LIN {X 0.002,Y -301.085,Z 1918.358,A 0.000,B 0.000,C 90.000,E1 64.357} C_DIS
LIN {X -0.093,Y -288.986,Z 1918.341,A 0.000,B 0.000,C 90.000,E1 61.385} C_DIS
LIN {X 0.024,Y -280.949,Z 1918.330,A 0.000,B 0.000,C 90.000,E1 59.331} C_DIS
LIN {X 0.071,Y -271.438,Z 1918.316,A 0.000,B 0.000,C 90.000,E1 56.914} C_DIS
LIN {X 0.067,Y -263.244,Z 1918.305,A 0.000,B 0.000,C 90.000,E1 54.815} C_DIS
LIN {X -0.054,Y -253.623,Z 1918.291,A 0.000,B 0.000,C 90.000,E1 52.351} C_DIS
LIN {X -0.111,Y -244.044,Z 1918.277,A 0.000,B 0.000,C 90.000,E1 49.828} C_DIS
LIN {X 0.069,Y -233.329,Z 1918.260,A 0.000,B 0.000,C 90.000,E1 46.824} C_DIS
LIN {X 0.121,Y -223.019,Z 1918.243,A 0.000,B 0.000,C 90.000,E1 43.785} C_DIS
LIN {X 0.001,Y -212.058,Z 1918.224,A 0.000,B 0.000,C 90.000,E1 40.334} C_DIS
LIN {X 0.010,Y -204.184,Z 1918.209,A 0.000,B 0.000,C 90.000,E1 37.569} C_DIS
LIN {X 0.020,Y -196.023,Z 1918.191,A 0.000,B 0.000,C 90.000,E1 34.358} C_DIS
LIN {X -0.106,Y -188.602,Z 1918.173,A 0.000,B 0.000,C 90.000,E1 31.131} C_DIS
LIN {X 0.030,Y -181.908,Z 1918.154,A 0.000,B 0.000,C 90.000,E1 27.769} C_DIS
LIN {X 0.067,Y -175.929,Z 1918.136,A 0.000,B 0.000,C 90.000,E1 24.387} C_DIS
LIN {X 0.063,Y -170.772,Z 1918.117,A 0.000,B 0.000,C 90.000,E1 20.972} C_DIS
LIN {X 0.072,Y -166.432,Z 1918.097,A 0.000,B 0.000,C 90.000,E1 17.511} C_DIS
LIN {X -0.056,Y -162.887,Z 1918.078,A 0.000,B 0.000,C 90.000,E1 14.064} C_DIS
LIN {X -0.062,Y -159.922,Z 1918.058,A 0.000,B 0.000,C 90.000,E1 10.546} C_DIS
LIN {X 0.005,Y -157.280,Z 1918.034,A 0.000,B 0.000,C 90.000,E1 6.087} C_DIS
LIN {X 0.000,Y -154.958,Z 1918.000,A 0.000,B 0.000,C 90.000,E1 360.000} C_DIS
LIN {X 0.053,Y -154.095,Z 1917.953,A 0.000,B 0.000,C 90.000,E1 351.432} C_DIS
LIN {X -0.028,Y -155.826,Z 1917.913,A 0.000,B 0.000,C 90.000,E1 344.283} C_DIS
LIN {X 0.033,Y -158.560,Z 1917.883,A 0.000,B 0.000,C 90.000,E1 338.901} C_DIS
LIN {X 0.047,Y -162.161,Z 1917.858,A 0.000,B 0.000,C 90.000,E1 334.460} C_DIS
LIN {X -0.046,Y -166.070,Z 1917.839,A 0.000,B 0.000,C 90.000,E1 330.973} C_DIS
LIN {X 0.051,Y -170.958,Z 1917.819,A 0.000,B 0.000,C 90.000,E1 327.454} C_DIS
LIN {X -0.037,Y -175.264,Z 1917.805,A 0.000,B 0.000,C 90.000,E1 324.895} C_DIS
LIN {X 0.017,Y -180.240,Z 1917.791,A 0.000,B 0.000,C 90.000,E1 322.316} C_DIS
LIN {X 0.016,Y -186.100,Z 1917.777,A 0.000,B 0.000,C 90.000,E1 319.784} C_DIS
LIN {X -0.018,Y -191.710,Z 1917.765,A 0.000,B 0.000,C 90.000,E1 317.715} C_DIS
LIN {X 0.020,Y -199.361,Z 1917.751,A 0.000,B 0.000,C 90.000,E1 315.243} C_DIS
LIN {X -0.078,Y -207.953,Z 1917.738,A 0.000,B 0.000,C 90.000,E1 312.852} C_DIS
LIN {X -0.098,Y -219.024,Z 1917.723,A 0.000,B 0.000,C 90.000,E1 310.092} C_DIS
LIN {X 0.025,Y -231.136,Z 1917.708,A 0.000,B 0.000,C 90.000,E1 307.363} C_DIS
LIN {X -0.158,Y -246.074,Z 1917.691,A 0.000,B 0.000,C 90.000,E1 304.405} C_DIS
LIN {X -0.153,Y -257.927,Z 1917.679,A 0.000,B 0.000,C 90.000,E1 302.212} C_DIS
LIN {X 0.088,Y -272.002,Z 1917.665,A 0.000,B 0.000,C 90.000,E1 299.667} C_DIS
LIN {X -0.137,Y -281.893,Z 1917.655,A 0.000,B 0.000,C 90.000,E1 297.975} C_DIS
LIN {X 0.036,Y -291.493,Z 1917.646,A 0.000,B 0.000,C 90.000,E1 296.232} C_DIS
LIN {X 0.116,Y -296.930,Z 1917.640,A 0.000,B 0.000,C 90.000,E1 295.207} C_DIS
LIN {X 0.120,Y -301.742,Z 1917.635,A 0.000,B 0.000,C 90.000,E1 294.207} C_DIS
LIN {X 0.005,Y -304.537,Z 1917.631,A 0.000,B 0.000,C 90.000,E1 293.567} C_DIS
LIN {X 0.067,Y -306.941,Z 1917.627,A 0.000,B 0.000,C 90.000,E1 292.898} C_DIS
LIN {X -0.019,Y -308.963,Z 1917.624,A 0.000,B 0.000,C 90.000,E1 292.259} C_DIS
LIN {X 0.070,Y -310.637,Z 1917.620,A 0.000,B 0.000,C 90.000,E1 291.589} C_DIS
LIN {X -0.116,Y -311.978,Z 1917.616,A 0.000,B 0.000,C 90.000,E1 290.972} C_DIS
LIN {X -0.001,Y -312.989,Z 1917.613,A 0.000,B 0.000,C 90.000,E1 290.301} C_DIS
LIN {X 0.124,Y -313.630,Z 1917.609,A 0.000,B 0.000,C 90.000,E1 289.631} C_DIS
LIN {X 0.145,Y -313.979,Z 1917.605,A 0.000,B 0.000,C 90.000,E1 288.960} C_DIS
LIN {X 0.090,Y -315.398,Z 1917.605,A 0.000,B 0.000,C 90.000,E1 288.960} C_DIS
LIN {X 0.111,Y -317.051,Z 1917.605,A 0.000,B 0.000,C 90.000,E1 288.906} C_DIS
LIN {X 0.074,Y -321.018,Z 1917.604,A 0.000,B 0.000,C 90.000,E1 288.671} C_DIS
LIN {X -0.008,Y -324.781,Z 1917.602,A 0.000,B 0.000,C 90.000,E1 288.362} C_DIS
LIN {X -0.038,Y -329.523,Z 1917.599,A 0.000,B 0.000,C 90.000,E1 287.873} C_DIS
LIN {X 0.007,Y -334.337,Z 1917.596,A 0.000,B 0.000,C 90.000,E1 287.275} C_DIS
LIN {X -0.155,Y -338.741,Z 1917.593,A 0.000,B 0.000,C 90.000,E1 286.677} C_DIS
LIN {X 0.038,Y -342.538,Z 1917.589,A 0.000,B 0.000,C 90.000,E1 286.024} C_DIS
LIN {X -0.073,Y -345.806,Z 1917.586,A 0.000,B 0.000,C 90.000,E1 285.426} C_DIS
LIN {X 0.173,Y -348.683,Z 1917.582,A 0.000,B 0.000,C 90.000,E1 284.773} C_DIS
LIN {X 0.027,Y -352.297,Z 1917.577,A 0.000,B 0.000,C 90.000,E1 283.883} C_DIS
LIN {X -0.172,Y -354.899,Z 1917.572,A 0.000,B 0.000,C 90.000,E1 283.008} C_DIS
LIN {X 0.132,Y -356.054,Z 1917.569,A 0.000,B 0.000,C 90.000,E1 282.355} C_DIS
LIN {X 0.021,Y -356.751,Z 1917.565,A 0.000,B 0.000,C 90.000,E1 281.771} C_DIS
LIN {X -0.083,Y -356.912,Z 1917.562,A 0.000,B 0.000,C 90.000,E1 281.186} C_DIS
LIN {X 0.169,Y -356.637,Z 1917.559,A 0.000,B 0.000,C 90.000,E1 280.546} C_DIS
LIN {X 0.070,Y -355.925,Z 1917.555,A 0.000,B 0.000,C 90.000,E1 279.962} C_DIS
LIN {X -0.032,Y -354.775,Z 1917.552,A 0.000,B 0.000,C 90.000,E1 279.378} C_DIS
LIN {X 0.155,Y -353.206,Z 1917.549,A 0.000,B 0.000,C 90.000,E1 278.746} C_DIS
LIN {X 0.041,Y -351.190,Z 1917.545,A 0.000,B 0.000,C 90.000,E1 278.163} C_DIS
LIN {X -0.132,Y -348.661,Z 1917.542,A 0.000,B 0.000,C 90.000,E1 277.587} C_DIS
LIN {X 0.066,Y -345.529,Z 1917.539,A 0.000,B 0.000,C 90.000,E1 276.947} C_DIS
LIN {X -0.056,Y -343.742,Z 1917.537,A 0.000,B 0.000,C 90.000,E1 276.663} C_DIS
LIN {X 0.071,Y -339.329,Z 1917.534,A 0.000,B 0.000,C 90.000,E1 276.030} C_DIS
LIN {X -0.022,Y -336.617,Z 1917.532,A 0.000,B 0.000,C 90.000,E1 275.739} C_DIS
LIN {X -0.082,Y -333.609,Z 1917.530,A 0.000,B 0.000,C 90.000,E1 275.448} C_DIS
LIN {X 0.158,Y -330.113,Z 1917.529,A 0.000,B 0.000,C 90.000,E1 275.106} C_DIS
LIN {X 0.053,Y -326.707,Z 1917.527,A 0.000,B 0.000,C 90.000,E1 274.878} C_DIS
LIN {X 0.082,Y -320.483,Z 1917.525,A 0.000,B 0.000,C 90.000,E1 274.531} C_DIS
LIN {X 0.041,Y -317.170,Z 1917.525,A 0.000,B 0.000,C 90.000,E1 274.416} C_DIS
LIN {X -0.141,Y -312.787,Z 1917.524,A 0.000,B 0.000,C 90.000,E1 274.359} C_DIS
LIN {X 0.063,Y -181.047,Z 1917.524,A 0.000,B 0.000,C 90.000,E1 274.302} C_DIS
LIN {X 0.057,Y -181.570,Z 1917.500,A 0.000,B 0.000,C 90.000,E1 270.057} C_DIS
LIN {X 0.044,Y -180.866,Z 1917.472,A 0.000,B 0.000,C 90.000,E1 265.008} C_DIS
LIN {X -0.078,Y -178.981,Z 1917.444,A 0.000,B 0.000,C 90.000,E1 259.982} C_DIS
LIN {X -0.067,Y -177.953,Z 1917.435,A 0.000,B 0.000,C 90.000,E1 258.285} C_DIS
LIN {X -0.048,Y -175.594,Z 1917.411,A 0.000,B 0.000,C 90.000,E1 254.031} C_DIS
LIN {X -0.035,Y -172.318,Z 1917.387,A 0.000,B 0.000,C 90.000,E1 249.752} C_DIS
LIN {X -0.056,Y -171.797,Z 1917.383,A 0.000,B 0.000,C 90.000,E1 248.901} C_DIS
LIN {X -0.019,Y -169.468,Z 1917.368,A 0.000,B 0.000,C 90.000,E1 246.305} C_DIS
LIN {X 0.037,Y -166.796,Z 1917.349,A 0.000,B 0.000,C 90.000,E1 242.820} C_DIS
LIN {X 0.032,Y -162.777,Z 1917.325,A 0.000,B 0.000,C 90.000,E1 238.456} C_DIS
LIN {X 0.008,Y -161.466,Z 1917.315,A 0.000,B 0.000,C 90.000,E1 236.707} C_DIS
LIN {X 0.049,Y -157.460,Z 1917.291,A 0.000,B 0.000,C 90.000,E1 232.271} C_DIS
LIN {X -0.018,Y -155.472,Z 1917.276,A 0.000,B 0.000,C 90.000,E1 229.622} C_DIS
LIN {X -0.085,Y -151.784,Z 1917.251,A 0.000,B 0.000,C 90.000,E1 225.162} C_DIS
LIN {X -0.071,Y -149.990,Z 1917.236,A 0.000,B 0.000,C 90.000,E1 222.447} C_DIS
LIN {X -0.040,Y -146.822,Z 1917.210,A 0.000,B 0.000,C 90.000,E1 217.890} C_DIS
LIN {X 0.066,Y -145.401,Z 1917.195,A 0.000,B 0.000,C 90.000,E1 215.105} C_DIS
LIN {X -0.017,Y -142.835,Z 1917.170,A 0.000,B 0.000,C 90.000,E1 210.541} C_DIS
LIN {X 0.040,Y -141.447,Z 1917.149,A 0.000,B 0.000,C 90.000,E1 206.821} C_DIS
LIN {X -0.047,Y -139.371,Z 1917.113,A 0.000,B 0.000,C 90.000,E1 200.355} C_DIS
LIN {X 0.070,Y -138.819,Z 1917.097,A 0.000,B 0.000,C 90.000,E1 197.511} C_DIS
LIN {X -0.016,Y -138.352,Z 1917.056,A 0.000,B 0.000,C 90.000,E1 190.074} C_DIS
LIN {X -0.043,Y -139.535,Z 1917.004,A 0.000,B 0.000,C 90.000,E1 180.745} C_DIS
LIN {X 0.051,Y -141.221,Z 1916.973,A 0.000,B 0.000,C 90.000,E1 175.122} C_DIS
LIN {X 0.009,Y -142.594,Z 1916.958,A 0.000,B 0.000,C 90.000,E1 172.356} C_DIS
LIN {X -0.038,Y -144.896,Z 1916.932,A 0.000,B 0.000,C 90.000,E1 167.757} C_DIS
LIN {X -0.084,Y -147.525,Z 1916.911,A 0.000,B 0.000,C 90.000,E1 164.102} C_DIS
LIN {X -0.010,Y -150.120,Z 1916.891,A 0.000,B 0.000,C 90.000,E1 160.423} C_DIS
LIN {X 0.001,Y -153.482,Z 1916.871,A 0.000,B 0.000,C 90.000,E1 156.794} C_DIS
LIN {X 0.065,Y -157.847,Z 1916.846,A 0.000,B 0.000,C 90.000,E1 152.281} C_DIS
LIN {X 0.021,Y -162.132,Z 1916.826,A 0.000,B 0.000,C 90.000,E1 148.742} C_DIS
LIN {X 0.000,Y -166.335,Z 1916.807,A 0.000,B 0.000,C 90.000,E1 145.229} C_DIS
LIN {X 0.007,Y -171.352,Z 1916.787,A 0.000,B 0.000,C 90.000,E1 141.743} C_DIS
LIN {X -0.066,Y -176.258,Z 1916.768,A 0.000,B 0.000,C 90.000,E1 138.324} C_DIS
LIN {X 0.052,Y -180.540,Z 1916.754,A 0.000,B 0.000,C 90.000,E1 135.729} C_DIS
LIN {X 0.032,Y -185.942,Z 1916.735,A 0.000,B 0.000,C 90.000,E1 132.366} C_DIS
LIN {X -0.033,Y -190.572,Z 1916.722,A 0.000,B 0.000,C 90.000,E1 129.886} C_DIS
LIN {X -0.003,Y -196.322,Z 1916.703,A 0.000,B 0.000,C 90.000,E1 126.583} C_DIS
LIN {X 0.075,Y -201.120,Z 1916.690,A 0.000,B 0.000,C 90.000,E1 124.119} C_DIS
LIN {X -0.006,Y -207.058,Z 1916.672,A 0.000,B 0.000,C 90.000,E1 120.924} C_DIS
LIN {X -0.010,Y -210.341,Z 1916.663,A 0.000,B 0.000,C 90.000,E1 119.333} C_DIS
LIN {X -0.016,Y -216.123,Z 1916.645,A 0.000,B 0.000,C 90.000,E1 116.181} C_DIS
LIN {X -0.112,Y -219.295,Z 1916.637,A 0.000,B 0.000,C 90.000,E1 114.643} C_DIS
LIN {X -0.109,Y -224.163,Z 1916.621,A 0.000,B 0.000,C 90.000,E1 111.844} C_DIS
LIN {X -0.174,Y -283.727,Z 1916.621,A 0.000,B 0.000,C 90.000,E1 111.844} C_DIS
LIN {X -0.106,Y -286.571,Z 1916.621,A 0.000,B 0.000,C 90.000,E1 111.770} C_DIS
LIN {X -0.081,Y -290.600,Z 1916.620,A 0.000,B 0.000,C 90.000,E1 111.535} C_DIS
LIN {X 0.088,Y -294.035,Z 1916.618,A 0.000,B 0.000,C 90.000,E1 111.153} C_DIS
LIN {X -0.092,Y -297.648,Z 1916.614,A 0.000,B 0.000,C 90.000,E1 110.610} C_DIS
LIN {X -0.075,Y -311.022,Z 1916.602,A 0.000,B 0.000,C 90.000,E1 108.290} C_DIS
LIN {X -0.041,Y -325.770,Z 1916.589,A 0.000,B 0.000,C 90.000,E1 106.024} C_DIS
LIN {X 0.046,Y -339.604,Z 1916.578,A 0.000,B 0.000,C 90.000,E1 104.120} C_DIS
LIN {X -0.103,Y -354.634,Z 1916.568,A 0.000,B 0.000,C 90.000,E1 102.299} C_DIS
LIN {X 0.070,Y -373.070,Z 1916.557,A 0.000,B 0.000,C 90.000,E1 100.254} C_DIS
LIN {X -0.187,Y -391.979,Z 1916.547,A 0.000,B 0.000,C 90.000,E1 98.454} C_DIS
LIN {X -0.144,Y -411.225,Z 1916.538,A 0.000,B 0.000,C 90.000,E1 96.777} C_DIS
LIN {X -0.198,Y -433.633,Z 1916.528,A 0.000,B 0.000,C 90.000,E1 95.049} C_DIS
LIN {X 0.220,Y -439.284,Z 1916.526,A 0.000,B 0.000,C 90.000,E1 94.588} C_DIS
LIN {X -0.005,Y -441.590,Z 1916.525,A 0.000,B 0.000,C 90.000,E1 94.416} C_DIS
LIN {X -0.020,Y -445.125,Z 1916.522,A 0.000,B 0.000,C 90.000,E1 93.955} C_DIS
LIN {X 0.154,Y -446.471,Z 1916.521,A 0.000,B 0.000,C 90.000,E1 93.669} C_DIS
LIN {X -0.117,Y -447.475,Z 1916.519,A 0.000,B 0.000,C 90.000,E1 93.440} C_DIS
LIN {X -0.159,Y -448.640,Z 1916.516,A 0.000,B 0.000,C 90.000,E1 92.922} C_DIS
LIN {X -0.219,Y -448.841,Z 1916.513,A 0.000,B 0.000,C 90.000,E1 92.407} C_DIS
LIN {X 0.181,Y -448.110,Z 1916.510,A 0.000,B 0.000,C 90.000,E1 91.835} C_DIS
LIN {X 0.145,Y -446.339,Z 1916.507,A 0.000,B 0.000,C 90.000,E1 91.318} C_DIS
LIN {X -0.104,Y -444.964,Z 1916.506,A 0.000,B 0.000,C 90.000,E1 91.088} C_DIS
LIN {X -0.166,Y -433.469,Z 1916.496,A 0.000,B 0.000,C 90.000,E1 89.255} C_DIS
LIN {X -0.150,Y -423.437,Z 1916.487,A 0.000,B 0.000,C 90.000,E1 87.650} C_DIS
LIN {X -0.195,Y -411.659,Z 1916.476,A 0.000,B 0.000,C 90.000,E1 85.755} C_DIS
LIN {X -0.129,Y -401.495,Z 1916.467,A 0.000,B 0.000,C 90.000,E1 84.090} C_DIS
LIN {X -0.151,Y -389.517,Z 1916.456,A 0.000,B 0.000,C 90.000,E1 82.129} C_DIS
LIN {X 0.064,Y -377.631,Z 1916.445,A 0.000,B 0.000,C 90.000,E1 80.095} C_DIS
LIN {X 0.039,Y -361.033,Z 1916.429,A 0.000,B 0.000,C 90.000,E1 77.173} C_DIS
LIN {X 0.113,Y -345.454,Z 1916.412,A 0.000,B 0.000,C 90.000,E1 74.157} C_DIS
LIN {X 0.041,Y -333.516,Z 1916.398,A 0.000,B 0.000,C 90.000,E1 71.710} C_DIS
LIN {X 0.042,Y -323.281,Z 1916.386,A 0.000,B 0.000,C 90.000,E1 69.518} C_DIS
LIN {X 0.114,Y -309.233,Z 1916.369,A 0.000,B 0.000,C 90.000,E1 66.305} C_DIS
LIN {X 0.062,Y -301.111,Z 1916.358,A 0.000,B 0.000,C 90.000,E1 64.357} C_DIS
LIN {X -0.034,Y -289.009,Z 1916.341,A 0.000,B 0.000,C 90.000,E1 61.385} C_DIS
LIN {X 0.082,Y -280.972,Z 1916.330,A 0.000,B 0.000,C 90.000,E1 59.331} C_DIS
LIN {X 0.128,Y -271.465,Z 1916.316,A 0.000,B 0.000,C 90.000,E1 56.914} C_DIS
LIN {X -0.029,Y -263.273,Z 1916.305,A 0.000,B 0.000,C 90.000,E1 54.848} C_DIS
LIN {X 0.000,Y -253.652,Z 1916.291,A 0.000,B 0.000,C 90.000,E1 52.351} C_DIS
LIN {X -0.059,Y -244.075,Z 1916.277,A 0.000,B 0.000,C 90.000,E1 49.828} C_DIS
LIN {X -0.040,Y -233.354,Z 1916.260,A 0.000,B 0.000,C 90.000,E1 46.863} C_DIS
LIN {X -0.145,Y -223.043,Z 1916.244,A 0.000,B 0.000,C 90.000,E1 43.866} C_DIS
LIN {X 0.048,Y -212.080,Z 1916.224,A 0.000,B 0.000,C 90.000,E1 40.334} C_DIS
LIN {X -0.068,Y -204.204,Z 1916.209,A 0.000,B 0.000,C 90.000,E1 37.604} C_DIS
LIN {X -0.097,Y -196.042,Z 1916.191,A 0.000,B 0.000,C 90.000,E1 34.405} C_DIS
LIN {X -0.063,Y -188.620,Z 1916.173,A 0.000,B 0.000,C 90.000,E1 31.131} C_DIS
LIN {X 0.073,Y -181.925,Z 1916.154,A 0.000,B 0.000,C 90.000,E1 27.769} C_DIS
LIN {X 0.108,Y -175.944,Z 1916.136,A 0.000,B 0.000,C 90.000,E1 24.387} C_DIS
LIN {X 0.103,Y -170.784,Z 1916.117,A 0.000,B 0.000,C 90.000,E1 20.972} C_DIS
LIN {X -0.097,Y -166.442,Z 1916.098,A 0.000,B 0.000,C 90.000,E1 17.583} C_DIS
LIN {X -0.017,Y -162.893,Z 1916.078,A 0.000,B 0.000,C 90.000,E1 14.064} C_DIS
LIN {X -0.024,Y -159.924,Z 1916.059,A 0.000,B 0.000,C 90.000,E1 10.546} C_DIS
LIN {X 0.044,Y -157.279,Z 1916.034,A 0.000,B 0.000,C 90.000,E1 6.087} C_DIS
LIN {X 0.000,Y -154.950,Z 1916.000,A 0.000,B 0.000,C 90.000,E1 360.000} C_DIS
LIN {X 0.053,Y -154.089,Z 1915.953,A 0.000,B 0.000,C 90.000,E1 351.432} C_DIS
LIN {X -0.029,Y -155.821,Z 1915.913,A 0.000,B 0.000,C 90.000,E1 344.283} C_DIS
LIN {X 0.032,Y -158.557,Z 1915.883,A 0.000,B 0.000,C 90.000,E1 338.901} C_DIS
LIN {X 0.046,Y -162.159,Z 1915.858,A 0.000,B 0.000,C 90.000,E1 334.460} C_DIS
LIN {X -0.047,Y -166.073,Z 1915.839,A 0.000,B 0.000,C 90.000,E1 330.973} C_DIS
LIN {X 0.050,Y -170.962,Z 1915.819,A 0.000,B 0.000,C 90.000,E1 327.454} C_DIS
LIN {X -0.037,Y -175.271,Z 1915.805,A 0.000,B 0.000,C 90.000,E1 324.895} C_DIS
LIN {X 0.016,Y -180.248,Z 1915.791,A 0.000,B 0.000,C 90.000,E1 322.316} C_DIS
LIN {X 0.015,Y -186.109,Z 1915.777,A 0.000,B 0.000,C 90.000,E1 319.784} C_DIS
LIN {X -0.019,Y -191.718,Z 1915.765,A 0.000,B 0.000,C 90.000,E1 317.715} C_DIS
LIN {X 0.020,Y -199.368,Z 1915.751,A 0.000,B 0.000,C 90.000,E1 315.243} C_DIS
LIN {X -0.078,Y -207.959,Z 1915.738,A 0.000,B 0.000,C 90.000,E1 312.852} C_DIS
LIN {X -0.098,Y -219.032,Z 1915.723,A 0.000,B 0.000,C 90.000,E1 310.092} C_DIS
LIN {X 0.025,Y -231.144,Z 1915.708,A 0.000,B 0.000,C 90.000,E1 307.363} C_DIS
LIN {X -0.157,Y -246.084,Z 1915.691,A 0.000,B 0.000,C 90.000,E1 304.405} C_DIS
LIN {X -0.152,Y -257.937,Z 1915.679,A 0.000,B 0.000,C 90.000,E1 302.212} C_DIS
LIN {X 0.089,Y -272.010,Z 1915.665,A 0.000,B 0.000,C 90.000,E1 299.667} C_DIS
LIN {X -0.137,Y -281.901,Z 1915.655,A 0.000,B 0.000,C 90.000,E1 297.975} C_DIS
LIN {X 0.036,Y -291.501,Z 1915.646,A 0.000,B 0.000,C 90.000,E1 296.232} C_DIS
LIN {X 0.118,Y -296.941,Z 1915.640,A 0.000,B 0.000,C 90.000,E1 295.207} C_DIS
LIN {X 0.121,Y -301.754,Z 1915.635,A 0.000,B 0.000,C 90.000,E1 294.207} C_DIS
LIN {X 0.006,Y -304.547,Z 1915.631,A 0.000,B 0.000,C 90.000,E1 293.567} C_DIS
LIN {X 0.068,Y -306.952,Z 1915.627,A 0.000,B 0.000,C 90.000,E1 292.898} C_DIS
LIN {X -0.018,Y -308.975,Z 1915.624,A 0.000,B 0.000,C 90.000,E1 292.259} C_DIS
LIN {X 0.071,Y -310.650,Z 1915.620,A 0.000,B 0.000,C 90.000,E1 291.589} C_DIS
LIN {X -0.114,Y -311.991,Z 1915.616,A 0.000,B 0.000,C 90.000,E1 290.972} C_DIS
LIN {X 0.091,Y -313.107,Z 1915.612,A 0.000,B 0.000,C 90.000,E1 290.194} C_DIS
LIN {X 0.035,Y -313.139,Z 1915.612,A 0.000,B 0.000,C 90.000,E1 290.194} C_DIS
LIN {X -0.084,Y -315.881,Z 1915.611,A 0.000,B 0.000,C 90.000,E1 289.993} C_DIS
LIN {X -0.046,Y -321.921,Z 1915.608,A 0.000,B 0.000,C 90.000,E1 289.396} C_DIS
LIN {X -0.102,Y -326.834,Z 1915.604,A 0.000,B 0.000,C 90.000,E1 288.833} C_DIS
LIN {X 0.076,Y -331.679,Z 1915.601,A 0.000,B 0.000,C 90.000,E1 288.181} C_DIS
LIN {X -0.102,Y -336.133,Z 1915.598,A 0.000,B 0.000,C 90.000,E1 287.583} C_DIS
LIN {X 0.172,Y -340.116,Z 1915.594,A 0.000,B 0.000,C 90.000,E1 286.913} C_DIS
LIN {X 0.047,Y -343.672,Z 1915.591,A 0.000,B 0.000,C 90.000,E1 286.315} C_DIS
LIN {X -0.151,Y -348.235,Z 1915.586,A 0.000,B 0.000,C 90.000,E1 285.426} C_DIS
LIN {X 0.038,Y -352.020,Z 1915.580,A 0.000,B 0.000,C 90.000,E1 284.481} C_DIS
LIN {X 0.052,Y -353.153,Z 1915.579,A 0.000,B 0.000,C 90.000,E1 284.175} C_DIS
LIN {X -0.080,Y -355.047,Z 1915.575,A 0.000,B 0.000,C 90.000,E1 283.592} C_DIS
LIN {X -0.203,Y -356.588,Z 1915.572,A 0.000,B 0.000,C 90.000,E1 283.008} C_DIS
LIN {X 0.114,Y -357.659,Z 1915.569,A 0.000,B 0.000,C 90.000,E1 282.355} C_DIS
LIN {X 0.012,Y -358.305,Z 1915.565,A 0.000,B 0.000,C 90.000,E1 281.771} C_DIS
LIN {X -0.082,Y -358.449,Z 1915.562,A 0.000,B 0.000,C 90.000,E1 281.186} C_DIS
LIN {X -0.172,Y -358.191,Z 1915.559,A 0.000,B 0.000,C 90.000,E1 280.602} C_DIS
LIN {X 0.090,Y -357.501,Z 1915.555,A 0.000,B 0.000,C 90.000,E1 279.962} C_DIS
LIN {X -0.003,Y -356.423,Z 1915.552,A 0.000,B 0.000,C 90.000,E1 279.378} C_DIS
LIN {X -0.156,Y -354.965,Z 1915.549,A 0.000,B 0.000,C 90.000,E1 278.803} C_DIS
LIN {X 0.032,Y -351.969,Z 1915.544,A 0.000,B 0.000,C 90.000,E1 277.871} C_DIS
LIN {X -0.140,Y -349.419,Z 1915.540,A 0.000,B 0.000,C 90.000,E1 277.296} C_DIS
LIN {X 0.020,Y -346.233,Z 1915.537,A 0.000,B 0.000,C 90.000,E1 276.663} C_DIS
LIN {X -0.179,Y -342.419,Z 1915.534,A 0.000,B 0.000,C 90.000,E1 276.087} C_DIS
LIN {X 0.075,Y -340.154,Z 1915.532,A 0.000,B 0.000,C 90.000,E1 275.739} C_DIS
LIN {X -0.153,Y -334.704,Z 1915.529,A 0.000,B 0.000,C 90.000,E1 275.163} C_DIS
LIN {X 0.143,Y -331.664,Z 1915.527,A 0.000,B 0.000,C 90.000,E1 274.821} C_DIS
LIN {X 0.133,Y -328.194,Z 1915.525,A 0.000,B 0.000,C 90.000,E1 274.531} C_DIS
LIN {X -0.020,Y -321.078,Z 1915.523,A 0.000,B 0.000,C 90.000,E1 274.073} C_DIS
LIN {X -0.114,Y -317.255,Z 1915.521,A 0.000,B 0.000,C 90.000,E1 273.898} C_DIS
LIN {X 0.029,Y -309.804,Z 1915.520,A 0.000,B 0.000,C 90.000,E1 273.612} C_DIS
LIN {X 0.013,Y -305.845,Z 1915.520,A 0.000,B 0.000,C 90.000,E1 273.555} C_DIS
LIN {X -0.028,Y -181.082,Z 1915.520,A 0.000,B 0.000,C 90.000,E1 273.555} C_DIS
LIN {X 0.060,Y -181.571,Z 1915.500,A 0.000,B 0.000,C 90.000,E1 270.057} C_DIS
LIN {X 0.048,Y -180.867,Z 1915.472,A 0.000,B 0.000,C 90.000,E1 265.008} C_DIS
LIN {X -0.075,Y -178.982,Z 1915.444,A 0.000,B 0.000,C 90.000,E1 259.982} C_DIS
LIN {X -0.063,Y -177.953,Z 1915.435,A 0.000,B 0.000,C 90.000,E1 258.285} C_DIS
LIN {X -0.044,Y -175.595,Z 1915.411,A 0.000,B 0.000,C 90.000,E1 254.031} C_DIS
LIN {X -0.031,Y -172.319,Z 1915.387,A 0.000,B 0.000,C 90.000,E1 249.752} C_DIS
LIN {X -0.052,Y -171.797,Z 1915.383,A 0.000,B 0.000,C 90.000,E1 248.901} C_DIS
LIN {X -0.015,Y -169.469,Z 1915.368,A 0.000,B 0.000,C 90.000,E1 246.305} C_DIS
LIN {X 0.040,Y -166.797,Z 1915.349,A 0.000,B 0.000,C 90.000,E1 242.820} C_DIS
LIN {X 0.035,Y -162.777,Z 1915.325,A 0.000,B 0.000,C 90.000,E1 238.456} C_DIS
LIN {X 0.011,Y -161.467,Z 1915.315,A 0.000,B 0.000,C 90.000,E1 236.707} C_DIS
LIN {X 0.052,Y -157.461,Z 1915.291,A 0.000,B 0.000,C 90.000,E1 232.271} C_DIS
LIN {X -0.015,Y -155.474,Z 1915.276,A 0.000,B 0.000,C 90.000,E1 229.622} C_DIS
LIN {X -0.081,Y -151.785,Z 1915.251,A 0.000,B 0.000,C 90.000,E1 225.162} C_DIS
LIN {X -0.069,Y -149.991,Z 1915.236,A 0.000,B 0.000,C 90.000,E1 222.447} C_DIS
LIN {X -0.037,Y -146.823,Z 1915.210,A 0.000,B 0.000,C 90.000,E1 217.890} C_DIS
LIN {X 0.069,Y -145.402,Z 1915.195,A 0.000,B 0.000,C 90.000,E1 215.105} C_DIS
LIN {X -0.014,Y -142.835,Z 1915.170,A 0.000,B 0.000,C 90.000,E1 210.541} C_DIS
LIN {X 0.043,Y -141.448,Z 1915.149,A 0.000,B 0.000,C 90.000,E1 206.821} C_DIS
LIN {X -0.044,Y -139.371,Z 1915.113,A 0.000,B 0.000,C 90.000,E1 200.355} C_DIS
LIN {X 0.073,Y -138.819,Z 1915.097,A 0.000,B 0.000,C 90.000,E1 197.511} C_DIS
LIN {X -0.013,Y -138.352,Z 1915.056,A 0.000,B 0.000,C 90.000,E1 190.074} C_DIS
LIN {X -0.040,Y -139.534,Z 1915.004,A 0.000,B 0.000,C 90.000,E1 180.745} C_DIS
LIN {X 0.053,Y -141.220,Z 1914.973,A 0.000,B 0.000,C 90.000,E1 175.122} C_DIS
LIN {X 0.012,Y -142.593,Z 1914.958,A 0.000,B 0.000,C 90.000,E1 172.356} C_DIS
LIN {X -0.034,Y -144.895,Z 1914.932,A 0.000,B 0.000,C 90.000,E1 167.757} C_DIS
LIN {X -0.081,Y -147.524,Z 1914.911,A 0.000,B 0.000,C 90.000,E1 164.102} C_DIS
LIN {X -0.007,Y -150.120,Z 1914.891,A 0.000,B 0.000,C 90.000,E1 160.423} C_DIS
LIN {X 0.004,Y -153.482,Z 1914.871,A 0.000,B 0.000,C 90.000,E1 156.794} C_DIS
LIN {X 0.068,Y -157.845,Z 1914.846,A 0.000,B 0.000,C 90.000,E1 152.281} C_DIS
LIN {X 0.024,Y -162.131,Z 1914.826,A 0.000,B 0.000,C 90.000,E1 148.742} C_DIS
LIN {X 0.004,Y -166.334,Z 1914.807,A 0.000,B 0.000,C 90.000,E1 145.229} C_DIS
LIN {X 0.010,Y -171.351,Z 1914.787,A 0.000,B 0.000,C 90.000,E1 141.743} C_DIS
LIN {X -0.063,Y -176.256,Z 1914.768,A 0.000,B 0.000,C 90.000,E1 138.324} C_DIS
LIN {X 0.056,Y -180.538,Z 1914.754,A 0.000,B 0.000,C 90.000,E1 135.729} C_DIS
LIN {X 0.036,Y -185.940,Z 1914.735,A 0.000,B 0.000,C 90.000,E1 132.366} C_DIS
LIN {X -0.029,Y -190.570,Z 1914.722,A 0.000,B 0.000,C 90.000,E1 129.886} C_DIS
LIN {X 0.001,Y -196.320,Z 1914.703,A 0.000,B 0.000,C 90.000,E1 126.583} C_DIS
LIN {X 0.078,Y -201.119,Z 1914.690,A 0.000,B 0.000,C 90.000,E1 124.119} C_DIS
LIN {X -0.002,Y -207.056,Z 1914.672,A 0.000,B 0.000,C 90.000,E1 120.924} C_DIS
LIN {X -0.007,Y -210.338,Z 1914.663,A 0.000,B 0.000,C 90.000,E1 119.333} C_DIS
LIN {X -0.013,Y -216.120,Z 1914.645,A 0.000,B 0.000,C 90.000,E1 116.181} C_DIS
LIN {X -0.108,Y -219.294,Z 1914.637,A 0.000,B 0.000,C 90.000,E1 114.643} C_DIS
LIN {X -0.106,Y -224.161,Z 1914.621,A 0.000,B 0.000,C 90.000,E1 111.844} C_DIS
LIN {X -0.168,Y -283.797,Z 1914.621,A 0.000,B 0.000,C 90.000,E1 111.844} C_DIS
LIN {X -0.101,Y -286.579,Z 1914.621,A 0.000,B 0.000,C 90.000,E1 111.770} C_DIS
LIN {X -0.076,Y -290.597,Z 1914.620,A 0.000,B 0.000,C 90.000,E1 111.535} C_DIS
LIN {X 0.089,Y -294.036,Z 1914.618,A 0.000,B 0.000,C 90.000,E1 111.153} C_DIS
LIN {X -0.093,Y -297.649,Z 1914.614,A 0.000,B 0.000,C 90.000,E1 110.610} C_DIS
LIN {X -0.078,Y -311.023,Z 1914.602,A 0.000,B 0.000,C 90.000,E1 108.290} C_DIS
LIN {X -0.042,Y -325.771,Z 1914.589,A 0.000,B 0.000,C 90.000,E1 106.024} C_DIS
LIN {X 0.044,Y -339.605,Z 1914.578,A 0.000,B 0.000,C 90.000,E1 104.120} C_DIS
LIN {X -0.106,Y -354.635,Z 1914.568,A 0.000,B 0.000,C 90.000,E1 102.299} C_DIS
LIN {X 0.067,Y -373.072,Z 1914.557,A 0.000,B 0.000,C 90.000,E1 100.254} C_DIS
LIN {X -0.188,Y -391.980,Z 1914.547,A 0.000,B 0.000,C 90.000,E1 98.454} C_DIS
LIN {X -0.145,Y -411.227,Z 1914.537,A 0.000,B 0.000,C 90.000,E1 96.777} C_DIS
LIN {X -0.199,Y -433.634,Z 1914.528,A 0.000,B 0.000,C 90.000,E1 95.049} C_DIS
LIN {X 0.219,Y -439.285,Z 1914.526,A 0.000,B 0.000,C 90.000,E1 94.588} C_DIS
LIN {X -0.007,Y -441.587,Z 1914.525,A 0.000,B 0.000,C 90.000,E1 94.416} C_DIS
LIN {X -0.026,Y -445.120,Z 1914.522,A 0.000,B 0.000,C 90.000,E1 93.955} C_DIS
LIN {X 0.148,Y -446.465,Z 1914.521,A 0.000,B 0.000,C 90.000,E1 93.669} C_DIS
LIN {X -0.124,Y -447.467,Z 1914.519,A 0.000,B 0.000,C 90.000,E1 93.440} C_DIS
LIN {X -0.165,Y -448.629,Z 1914.516,A 0.000,B 0.000,C 90.000,E1 92.922} C_DIS
LIN {X -0.224,Y -448.827,Z 1914.513,A 0.000,B 0.000,C 90.000,E1 92.407} C_DIS
LIN {X 0.174,Y -448.093,Z 1914.510,A 0.000,B 0.000,C 90.000,E1 91.835} C_DIS
LIN {X 0.138,Y -446.318,Z 1914.507,A 0.000,B 0.000,C 90.000,E1 91.318} C_DIS
LIN {X -0.110,Y -444.941,Z 1914.506,A 0.000,B 0.000,C 90.000,E1 91.088} C_DIS
LIN {X -0.174,Y -433.444,Z 1914.496,A 0.000,B 0.000,C 90.000,E1 89.255} C_DIS
LIN {X -0.157,Y -423.413,Z 1914.487,A 0.000,B 0.000,C 90.000,E1 87.650} C_DIS
LIN {X 0.209,Y -411.634,Z 1914.476,A 0.000,B 0.000,C 90.000,E1 85.698} C_DIS
LIN {X -0.135,Y -401.470,Z 1914.467,A 0.000,B 0.000,C 90.000,E1 84.090} C_DIS
LIN {X -0.160,Y -389.493,Z 1914.456,A 0.000,B 0.000,C 90.000,E1 82.129} C_DIS
LIN {X 0.055,Y -377.607,Z 1914.445,A 0.000,B 0.000,C 90.000,E1 80.095} C_DIS
LIN {X 0.031,Y -361.006,Z 1914.429,A 0.000,B 0.000,C 90.000,E1 77.173} C_DIS
LIN {X 0.103,Y -345.428,Z 1914.412,A 0.000,B 0.000,C 90.000,E1 74.157} C_DIS
LIN {X 0.032,Y -333.489,Z 1914.398,A 0.000,B 0.000,C 90.000,E1 71.710} C_DIS
LIN {X 0.033,Y -323.253,Z 1914.386,A 0.000,B 0.000,C 90.000,E1 69.518} C_DIS
LIN {X 0.104,Y -309.205,Z 1914.368,A 0.000,B 0.000,C 90.000,E1 66.305} C_DIS
LIN {X 0.052,Y -301.082,Z 1914.358,A 0.000,B 0.000,C 90.000,E1 64.357} C_DIS
LIN {X -0.045,Y -288.978,Z 1914.341,A 0.000,B 0.000,C 90.000,E1 61.385} C_DIS
LIN {X 0.071,Y -280.940,Z 1914.330,A 0.000,B 0.000,C 90.000,E1 59.331} C_DIS
LIN {X 0.116,Y -271.436,Z 1914.316,A 0.000,B 0.000,C 90.000,E1 56.914} C_DIS
LIN {X -0.041,Y -263.245,Z 1914.305,A 0.000,B 0.000,C 90.000,E1 54.848} C_DIS
LIN {X -0.012,Y -253.625,Z 1914.291,A 0.000,B 0.000,C 90.000,E1 52.351} C_DIS
LIN {X -0.071,Y -244.047,Z 1914.277,A 0.000,B 0.000,C 90.000,E1 49.828} C_DIS
LIN {X -0.052,Y -233.326,Z 1914.260,A 0.000,B 0.000,C 90.000,E1 46.863} C_DIS
LIN {X 0.004,Y -223.015,Z 1914.244,A 0.000,B 0.000,C 90.000,E1 43.824} C_DIS
LIN {X 0.036,Y -212.053,Z 1914.224,A 0.000,B 0.000,C 90.000,E1 40.334} C_DIS
LIN {X -0.081,Y -204.181,Z 1914.209,A 0.000,B 0.000,C 90.000,E1 37.604} C_DIS
LIN {X -0.109,Y -196.023,Z 1914.191,A 0.000,B 0.000,C 90.000,E1 34.405} C_DIS
LIN {X -0.075,Y -188.603,Z 1914.173,A 0.000,B 0.000,C 90.000,E1 31.131} C_DIS
LIN {X 0.060,Y -181.909,Z 1914.154,A 0.000,B 0.000,C 90.000,E1 27.769} C_DIS
LIN {X 0.096,Y -175.930,Z 1914.136,A 0.000,B 0.000,C 90.000,E1 24.387} C_DIS
LIN {X 0.091,Y -170.774,Z 1914.117,A 0.000,B 0.000,C 90.000,E1 20.972} C_DIS
LIN {X 0.050,Y -166.431,Z 1914.098,A 0.000,B 0.000,C 90.000,E1 17.528} C_DIS
LIN {X -0.029,Y -162.881,Z 1914.078,A 0.000,B 0.000,C 90.000,E1 14.064} C_DIS
LIN {X -0.036,Y -159.913,Z 1914.058,A 0.000,B 0.000,C 90.000,E1 10.546} C_DIS
LIN {X 0.030,Y -157.270,Z 1914.034,A 0.000,B 0.000,C 90.000,E1 6.087} C_DIS
LIN {X 0.000,Y -154.941,Z 1914.000,A 0.000,B 0.000,C 90.000,E1 360.000} C_DIS
LIN {X -0.009,Y -154.159,Z 1913.948,A 0.000,B 0.000,C 90.000,E1 350.557} C_DIS
LIN {X -0.003,Y -156.156,Z 1913.908,A 0.000,B 0.000,C 90.000,E1 343.378} C_DIS
LIN {X 0.032,Y -158.555,Z 1913.883,A 0.000,B 0.000,C 90.000,E1 338.901} C_DIS
LIN {X 0.045,Y -162.157,Z 1913.858,A 0.000,B 0.000,C 90.000,E1 334.460} C_DIS
LIN {X -0.048,Y -166.076,Z 1913.839,A 0.000,B 0.000,C 90.000,E1 330.973} C_DIS
LIN {X 0.050,Y -170.967,Z 1913.819,A 0.000,B 0.000,C 90.000,E1 327.454} C_DIS
LIN {X -0.039,Y -175.278,Z 1913.805,A 0.000,B 0.000,C 90.000,E1 324.895} C_DIS
LIN {X 0.015,Y -180.256,Z 1913.791,A 0.000,B 0.000,C 90.000,E1 322.316} C_DIS
LIN {X 0.014,Y -186.117,Z 1913.777,A 0.000,B 0.000,C 90.000,E1 319.784} C_DIS
LIN {X -0.019,Y -191.725,Z 1913.765,A 0.000,B 0.000,C 90.000,E1 317.715} C_DIS
LIN {X 0.019,Y -199.374,Z 1913.751,A 0.000,B 0.000,C 90.000,E1 315.243} C_DIS
LIN {X -0.079,Y -207.966,Z 1913.738,A 0.000,B 0.000,C 90.000,E1 312.852} C_DIS
LIN {X -0.098,Y -219.040,Z 1913.723,A 0.000,B 0.000,C 90.000,E1 310.092} C_DIS
LIN {X 0.025,Y -231.153,Z 1913.708,A 0.000,B 0.000,C 90.000,E1 307.363} C_DIS
LIN {X -0.157,Y -246.094,Z 1913.691,A 0.000,B 0.000,C 90.000,E1 304.405} C_DIS
LIN {X -0.152,Y -257.946,Z 1913.679,A 0.000,B 0.000,C 90.000,E1 302.212} C_DIS
LIN {X 0.090,Y -272.019,Z 1913.665,A 0.000,B 0.000,C 90.000,E1 299.667} C_DIS
LIN {X -0.136,Y -281.910,Z 1913.655,A 0.000,B 0.000,C 90.000,E1 297.975} C_DIS
LIN {X 0.037,Y -291.511,Z 1913.646,A 0.000,B 0.000,C 90.000,E1 296.232} C_DIS
LIN {X 0.119,Y -296.953,Z 1913.640,A 0.000,B 0.000,C 90.000,E1 295.207} C_DIS
LIN {X 0.121,Y -301.766,Z 1913.635,A 0.000,B 0.000,C 90.000,E1 294.207} C_DIS
LIN {X 0.007,Y -304.557,Z 1913.631,A 0.000,B 0.000,C 90.000,E1 293.567} C_DIS
LIN {X 0.069,Y -306.963,Z 1913.627,A 0.000,B 0.000,C 90.000,E1 292.898} C_DIS
LIN {X -0.016,Y -308.988,Z 1913.624,A 0.000,B 0.000,C 90.000,E1 292.259} C_DIS
LIN {X -0.019,Y -311.348,Z 1913.618,A 0.000,B 0.000,C 90.000,E1 291.280} C_DIS
LIN {X 0.093,Y -311.791,Z 1913.617,A 0.000,B 0.000,C 90.000,E1 291.046} C_DIS
LIN {X 0.038,Y -311.852,Z 1913.617,A 0.000,B 0.000,C 90.000,E1 291.046} C_DIS
LIN {X 0.069,Y -315.578,Z 1913.615,A 0.000,B 0.000,C 90.000,E1 290.663} C_DIS
LIN {X -0.115,Y -320.644,Z 1913.612,A 0.000,B 0.000,C 90.000,E1 290.120} C_DIS
LIN {X 0.173,Y -325.622,Z 1913.608,A 0.000,B 0.000,C 90.000,E1 289.450} C_DIS
LIN {X -0.087,Y -332.485,Z 1913.603,A 0.000,B 0.000,C 90.000,E1 288.544} C_DIS
LIN {X 0.040,Y -338.636,Z 1913.598,A 0.000,B 0.000,C 90.000,E1 287.583} C_DIS
LIN {X -0.104,Y -343.960,Z 1913.593,A 0.000,B 0.000,C 90.000,E1 286.677} C_DIS
LIN {X 0.134,Y -348.469,Z 1913.587,A 0.000,B 0.000,C 90.000,E1 285.717} C_DIS
LIN {X -0.018,Y -352.296,Z 1913.582,A 0.000,B 0.000,C 90.000,E1 284.828} C_DIS
LIN {X -0.158,Y -354.489,Z 1913.579,A 0.000,B 0.000,C 90.000,E1 284.245} C_DIS
LIN {X 0.150,Y -356.297,Z 1913.576,A 0.000,B 0.000,C 90.000,E1 283.592} C_DIS
LIN {X 0.036,Y -357.783,Z 1913.572,A 0.000,B 0.000,C 90.000,E1 283.008} C_DIS
LIN {X 0.011,Y -358.821,Z 1913.569,A 0.000,B 0.000,C 90.000,E1 282.411} C_DIS
LIN {X -0.084,Y -359.459,Z 1913.566,A 0.000,B 0.000,C 90.000,E1 281.827} C_DIS
LIN {X 0.180,Y -359.628,Z 1913.562,A 0.000,B 0.000,C 90.000,E1 281.186} C_DIS
LIN {X 0.097,Y -359.406,Z 1913.559,A 0.000,B 0.000,C 90.000,E1 280.602} C_DIS
LIN {X 0.013,Y -358.740,Z 1913.556,A 0.000,B 0.000,C 90.000,E1 280.018} C_DIS
LIN {X -0.072,Y -357.742,Z 1913.552,A 0.000,B 0.000,C 90.000,E1 279.434} C_DIS
LIN {X 0.133,Y -356.388,Z 1913.549,A 0.000,B 0.000,C 90.000,E1 278.803} C_DIS
LIN {X 0.035,Y -354.600,Z 1913.546,A 0.000,B 0.000,C 90.000,E1 278.219} C_DIS
LIN {X 0.169,Y -351.196,Z 1913.541,A 0.000,B 0.000,C 90.000,E1 277.296} C_DIS
LIN {X -0.076,Y -346.660,Z 1913.536,A 0.000,B 0.000,C 90.000,E1 276.429} C_DIS
LIN {X 0.068,Y -342.806,Z 1913.532,A 0.000,B 0.000,C 90.000,E1 275.796} C_DIS
LIN {X -0.148,Y -338.043,Z 1913.529,A 0.000,B 0.000,C 90.000,E1 275.220} C_DIS
LIN {X -0.052,Y -332.227,Z 1913.525,A 0.000,B 0.000,C 90.000,E1 274.588} C_DIS
LIN {X 0.066,Y -325.704,Z 1913.522,A 0.000,B 0.000,C 90.000,E1 274.012} C_DIS
LIN {X 0.038,Y -322.504,Z 1913.521,A 0.000,B 0.000,C 90.000,E1 273.784} C_DIS
LIN {X -0.068,Y -315.226,Z 1913.519,A 0.000,B 0.000,C 90.000,E1 273.383} C_DIS
LIN {X 0.072,Y -308.711,Z 1913.517,A 0.000,B 0.000,C 90.000,E1 273.094} C_DIS
LIN {X 0.142,Y -304.896,Z 1913.517,A 0.000,B 0.000,C 90.000,E1 272.980} C_DIS
LIN {X 0.039,Y -299.187,Z 1913.516,A 0.000,B 0.000,C 90.000,E1 272.922} C_DIS
LIN {X 0.005,Y -181.137,Z 1913.516,A 0.000,B 0.000,C 90.000,E1 272.922} C_DIS
LIN {X -0.031,Y -181.567,Z 1913.500,A 0.000,B 0.000,C 90.000,E1 270.057} C_DIS
LIN {X -0.043,Y -180.861,Z 1913.472,A 0.000,B 0.000,C 90.000,E1 265.008} C_DIS
LIN {X 0.010,Y -178.974,Z 1913.444,A 0.000,B 0.000,C 90.000,E1 259.926} C_DIS
LIN {X 0.021,Y -177.934,Z 1913.435,A 0.000,B 0.000,C 90.000,E1 258.229} C_DIS
LIN {X 0.035,Y -175.573,Z 1913.411,A 0.000,B 0.000,C 90.000,E1 253.976} C_DIS
LIN {X 0.042,Y -172.300,Z 1913.387,A 0.000,B 0.000,C 90.000,E1 249.699} C_DIS
LIN {X 0.019,Y -171.779,Z 1913.383,A 0.000,B 0.000,C 90.000,E1 248.847} C_DIS
LIN {X -0.008,Y -168.709,Z 1913.363,A 0.000,B 0.000,C 90.000,E1 245.409} C_DIS
LIN {X 0.030,Y -166.773,Z 1913.349,A 0.000,B 0.000,C 90.000,E1 242.794} C_DIS
LIN {X -0.050,Y -162.754,Z 1913.325,A 0.000,B 0.000,C 90.000,E1 238.456} C_DIS
LIN {X -0.074,Y -161.443,Z 1913.315,A 0.000,B 0.000,C 90.000,E1 236.707} C_DIS
LIN {X -0.031,Y -157.437,Z 1913.290,A 0.000,B 0.000,C 90.000,E1 232.271} C_DIS
LIN {X 0.003,Y -155.445,Z 1913.276,A 0.000,B 0.000,C 90.000,E1 229.585} C_DIS
LIN {X 0.051,Y -151.764,Z 1913.251,A 0.000,B 0.000,C 90.000,E1 225.081} C_DIS
LIN {X 0.062,Y -149.966,Z 1913.235,A 0.000,B 0.000,C 90.000,E1 222.366} C_DIS
LIN {X -0.027,Y -146.805,Z 1913.210,A 0.000,B 0.000,C 90.000,E1 217.855} C_DIS
LIN {X -0.011,Y -145.381,Z 1913.195,A 0.000,B 0.000,C 90.000,E1 215.105} C_DIS
LIN {X -0.018,Y -142.441,Z 1913.164,A 0.000,B 0.000,C 90.000,E1 209.589} C_DIS
LIN {X 0.028,Y -141.433,Z 1913.149,A 0.000,B 0.000,C 90.000,E1 206.796} C_DIS
LIN {X 0.010,Y -139.366,Z 1913.113,A 0.000,B 0.000,C 90.000,E1 200.301} C_DIS
LIN {X -0.004,Y -138.811,Z 1913.097,A 0.000,B 0.000,C 90.000,E1 197.511} C_DIS
LIN {X 0.047,Y -138.351,Z 1913.056,A 0.000,B 0.000,C 90.000,E1 190.018} C_DIS
LIN {X 0.023,Y -139.540,Z 1913.004,A 0.000,B 0.000,C 90.000,E1 180.688} C_DIS
LIN {X -0.025,Y -141.235,Z 1912.973,A 0.000,B 0.000,C 90.000,E1 175.122} C_DIS
LIN {X -0.067,Y -142.605,Z 1912.957,A 0.000,B 0.000,C 90.000,E1 172.356} C_DIS
LIN {X 0.028,Y -144.915,Z 1912.932,A 0.000,B 0.000,C 90.000,E1 167.701} C_DIS
LIN {X 0.021,Y -147.544,Z 1912.911,A 0.000,B 0.000,C 90.000,E1 164.031} C_DIS
LIN {X 0.053,Y -150.145,Z 1912.891,A 0.000,B 0.000,C 90.000,E1 160.369} C_DIS
LIN {X 0.063,Y -153.514,Z 1912.871,A 0.000,B 0.000,C 90.000,E1 156.741} C_DIS
LIN {X -0.016,Y -157.879,Z 1912.846,A 0.000,B 0.000,C 90.000,E1 152.281} C_DIS
LIN {X -0.061,Y -162.166,Z 1912.826,A 0.000,B 0.000,C 90.000,E1 148.742} C_DIS
LIN {X 0.054,Y -166.374,Z 1912.807,A 0.000,B 0.000,C 90.000,E1 145.182} C_DIS
LIN {X 0.057,Y -171.390,Z 1912.787,A 0.000,B 0.000,C 90.000,E1 141.698} C_DIS
LIN {X 0.096,Y -176.301,Z 1912.768,A 0.000,B 0.000,C 90.000,E1 138.243} C_DIS
LIN {X -0.035,Y -180.588,Z 1912.754,A 0.000,B 0.000,C 90.000,E1 135.729} C_DIS
LIN {X -0.057,Y -185.990,Z 1912.735,A 0.000,B 0.000,C 90.000,E1 132.366} C_DIS
LIN {X -0.002,Y -190.623,Z 1912.721,A 0.000,B 0.000,C 90.000,E1 129.850} C_DIS
LIN {X -0.095,Y -196.374,Z 1912.703,A 0.000,B 0.000,C 90.000,E1 126.583} C_DIS
LIN {X -0.019,Y -201.165,Z 1912.690,A 0.000,B 0.000,C 90.000,E1 124.119} C_DIS
LIN {X 0.077,Y -207.111,Z 1912.672,A 0.000,B 0.000,C 90.000,E1 120.875} C_DIS
LIN {X 0.078,Y -210.388,Z 1912.663,A 0.000,B 0.000,C 90.000,E1 119.283} C_DIS
LIN {X -0.019,Y -216.174,Z 1912.645,A 0.000,B 0.000,C 90.000,E1 116.155} C_DIS
LIN {X -0.010,Y -219.341,Z 1912.637,A 0.000,B 0.000,C 90.000,E1 114.591} C_DIS
LIN {X -0.081,Y -224.150,Z 1912.621,A 0.000,B 0.000,C 90.000,E1 111.844} C_DIS
LIN {X -0.154,Y -283.627,Z 1912.621,A 0.000,B 0.000,C 90.000,E1 111.844} C_DIS
LIN {X 0.111,Y -285.137,Z 1912.621,A 0.000,B 0.000,C 90.000,E1 111.770} C_DIS
LIN {X 0.061,Y -290.930,Z 1912.619,A 0.000,B 0.000,C 90.000,E1 111.482} C_DIS
LIN {X 0.012,Y -293.993,Z 1912.618,A 0.000,B 0.000,C 90.000,E1 111.173} C_DIS
LIN {X -0.110,Y -297.665,Z 1912.614,A 0.000,B 0.000,C 90.000,E1 110.610} C_DIS
LIN {X -0.095,Y -311.041,Z 1912.602,A 0.000,B 0.000,C 90.000,E1 108.290} C_DIS
LIN {X -0.060,Y -325.792,Z 1912.589,A 0.000,B 0.000,C 90.000,E1 106.024} C_DIS
LIN {X 0.026,Y -339.627,Z 1912.578,A 0.000,B 0.000,C 90.000,E1 104.120} C_DIS
LIN {X -0.124,Y -354.660,Z 1912.568,A 0.000,B 0.000,C 90.000,E1 102.299} C_DIS
LIN {X 0.049,Y -373.097,Z 1912.557,A 0.000,B 0.000,C 90.000,E1 100.254} C_DIS
LIN {X -0.206,Y -392.005,Z 1912.547,A 0.000,B 0.000,C 90.000,E1 98.454} C_DIS
LIN {X -0.163,Y -411.253,Z 1912.537,A 0.000,B 0.000,C 90.000,E1 96.777} C_DIS
LIN {X -0.216,Y -433.662,Z 1912.528,A 0.000,B 0.000,C 90.000,E1 95.049} C_DIS
LIN {X 0.203,Y -439.311,Z 1912.526,A 0.000,B 0.000,C 90.000,E1 94.588} C_DIS
LIN {X -0.023,Y -441.601,Z 1912.525,A 0.000,B 0.000,C 90.000,E1 94.416} C_DIS
LIN {X -0.052,Y -445.131,Z 1912.522,A 0.000,B 0.000,C 90.000,E1 93.955} C_DIS
LIN {X 0.121,Y -446.469,Z 1912.521,A 0.000,B 0.000,C 90.000,E1 93.669} C_DIS
LIN {X -0.151,Y -447.466,Z 1912.519,A 0.000,B 0.000,C 90.000,E1 93.440} C_DIS
LIN {X -0.192,Y -448.621,Z 1912.516,A 0.000,B 0.000,C 90.000,E1 92.922} C_DIS
LIN {X 0.197,Y -448.811,Z 1912.513,A 0.000,B 0.000,C 90.000,E1 92.350} C_DIS
LIN {X 0.148,Y -448.069,Z 1912.510,A 0.000,B 0.000,C 90.000,E1 91.835} C_DIS
LIN {X 0.111,Y -446.285,Z 1912.507,A 0.000,B 0.000,C 90.000,E1 91.318} C_DIS
LIN {X -0.138,Y -444.902,Z 1912.506,A 0.000,B 0.000,C 90.000,E1 91.088} C_DIS
LIN {X -0.046,Y -431.759,Z 1912.494,A 0.000,B 0.000,C 90.000,E1 88.969} C_DIS
LIN {X 0.055,Y -420.004,Z 1912.484,A 0.000,B 0.000,C 90.000,E1 87.078} C_DIS
LIN {X -0.039,Y -408.217,Z 1912.473,A 0.000,B 0.000,C 90.000,E1 85.179} C_DIS
LIN {X 0.041,Y -396.305,Z 1912.462,A 0.000,B 0.000,C 90.000,E1 83.223} C_DIS
LIN {X -0.058,Y -382.648,Z 1912.450,A 0.000,B 0.000,C 90.000,E1 80.971} C_DIS
LIN {X 0.082,Y -369.150,Z 1912.437,A 0.000,B 0.000,C 90.000,E1 78.634} C_DIS
LIN {X -0.112,Y -353.043,Z 1912.420,A 0.000,B 0.000,C 90.000,E1 75.700} C_DIS
LIN {X -0.085,Y -339.377,Z 1912.405,A 0.000,B 0.000,C 90.000,E1 72.960} C_DIS
LIN {X -0.084,Y -327.585,Z 1912.391,A 0.000,B 0.000,C 90.000,E1 70.477} C_DIS
LIN {X -0.028,Y -314.678,Z 1912.376,A 0.000,B 0.000,C 90.000,E1 67.614} C_DIS
LIN {X -0.039,Y -303.758,Z 1912.361,A 0.000,B 0.000,C 90.000,E1 65.025} C_DIS
LIN {X 0.084,Y -292.901,Z 1912.347,A 0.000,B 0.000,C 90.000,E1 62.359} C_DIS
LIN {X 0.130,Y -284.943,Z 1912.335,A 0.000,B 0.000,C 90.000,E1 60.333} C_DIS
LIN {X -0.073,Y -276.828,Z 1912.324,A 0.000,B 0.000,C 90.000,E1 58.329} C_DIS
LIN {X 0.027,Y -267.322,Z 1912.310,A 0.000,B 0.000,C 90.000,E1 55.881} C_DIS
LIN {X -0.003,Y -257.693,Z 1912.297,A 0.000,B 0.000,C 90.000,E1 53.417} C_DIS
LIN {X 0.060,Y -248.100,Z 1912.283,A 0.000,B 0.000,C 90.000,E1 50.884} C_DIS
LIN {X 0.015,Y -237.255,Z 1912.266,A 0.000,B 0.000,C 90.000,E1 47.957} C_DIS
LIN {X 0.002,Y -226.802,Z 1912.250,A 0.000,B 0.000,C 90.000,E1 44.960} C_DIS
LIN {X -0.031,Y -215.575,Z 1912.231,A 0.000,B 0.000,C 90.000,E1 41.515} C_DIS
LIN {X -0.053,Y -206.332,Z 1912.213,A 0.000,B 0.000,C 90.000,E1 38.382} C_DIS
LIN {X -0.040,Y -197.984,Z 1912.195,A 0.000,B 0.000,C 90.000,E1 35.185} C_DIS
LIN {X -0.016,Y -190.367,Z 1912.177,A 0.000,B 0.000,C 90.000,E1 31.926} C_DIS
LIN {X -0.001,Y -183.507,Z 1912.159,A 0.000,B 0.000,C 90.000,E1 28.615} C_DIS
LIN {X -0.081,Y -177.326,Z 1912.140,A 0.000,B 0.000,C 90.000,E1 25.283} C_DIS
LIN {X 0.024,Y -171.979,Z 1912.121,A 0.000,B 0.000,C 90.000,E1 21.844} C_DIS
LIN {X -0.036,Y -167.414,Z 1912.102,A 0.000,B 0.000,C 90.000,E1 18.417} C_DIS
LIN {X 0.065,Y -163.690,Z 1912.083,A 0.000,B 0.000,C 90.000,E1 14.898} C_DIS
LIN {X -0.061,Y -159.898,Z 1912.058,A 0.000,B 0.000,C 90.000,E1 10.546} C_DIS
LIN {X 0.006,Y -157.258,Z 1912.034,A 0.000,B 0.000,C 90.000,E1 6.087} C_DIS
LIN {X 0.000,Y -154.933,Z 1912.000,A 0.000,B 0.000,C 90.000,E1 360.000} C_DIS
LIN {X -0.009,Y -154.152,Z 1911.948,A 0.000,B 0.000,C 90.000,E1 350.557} C_DIS
LIN {X -0.004,Y -156.152,Z 1911.908,A 0.000,B 0.000,C 90.000,E1 343.378} C_DIS
LIN {X 0.030,Y -158.553,Z 1911.883,A 0.000,B 0.000,C 90.000,E1 338.901} C_DIS
LIN {X 0.044,Y -162.157,Z 1911.858,A 0.000,B 0.000,C 90.000,E1 334.460} C_DIS
LIN {X -0.049,Y -166.078,Z 1911.839,A 0.000,B 0.000,C 90.000,E1 330.973} C_DIS
LIN {X 0.048,Y -170.971,Z 1911.819,A 0.000,B 0.000,C 90.000,E1 327.454} C_DIS
LIN {X -0.039,Y -175.284,Z 1911.805,A 0.000,B 0.000,C 90.000,E1 324.895} C_DIS
LIN {X 0.014,Y -180.264,Z 1911.791,A 0.000,B 0.000,C 90.000,E1 322.316} C_DIS
LIN {X 0.014,Y -186.127,Z 1911.777,A 0.000,B 0.000,C 90.000,E1 319.784} C_DIS
LIN {X -0.020,Y -191.733,Z 1911.765,A 0.000,B 0.000,C 90.000,E1 317.715} C_DIS
LIN {X 0.019,Y -199.380,Z 1911.751,A 0.000,B 0.000,C 90.000,E1 315.243} C_DIS
LIN {X -0.079,Y -207.972,Z 1911.738,A 0.000,B 0.000,C 90.000,E1 312.852} C_DIS
LIN {X -0.099,Y -219.048,Z 1911.723,A 0.000,B 0.000,C 90.000,E1 310.092} C_DIS
LIN {X 0.024,Y -231.161,Z 1911.708,A 0.000,B 0.000,C 90.000,E1 307.363} C_DIS
LIN {X -0.157,Y -246.104,Z 1911.691,A 0.000,B 0.000,C 90.000,E1 304.405} C_DIS
LIN {X -0.151,Y -257.956,Z 1911.679,A 0.000,B 0.000,C 90.000,E1 302.212} C_DIS
LIN {X 0.090,Y -272.027,Z 1911.665,A 0.000,B 0.000,C 90.000,E1 299.667} C_DIS
LIN {X -0.135,Y -281.919,Z 1911.655,A 0.000,B 0.000,C 90.000,E1 297.975} C_DIS
LIN {X 0.038,Y -291.520,Z 1911.646,A 0.000,B 0.000,C 90.000,E1 296.232} C_DIS
LIN {X 0.120,Y -296.964,Z 1911.640,A 0.000,B 0.000,C 90.000,E1 295.207} C_DIS
LIN {X 0.123,Y -301.775,Z 1911.635,A 0.000,B 0.000,C 90.000,E1 294.207} C_DIS
LIN {X 0.008,Y -304.566,Z 1911.631,A 0.000,B 0.000,C 90.000,E1 293.567} C_DIS
LIN {X -0.030,Y -308.035,Z 1911.625,A 0.000,B 0.000,C 90.000,E1 292.589} C_DIS
LIN {X 0.096,Y -310.227,Z 1911.621,A 0.000,B 0.000,C 90.000,E1 291.770} C_DIS
LIN {X 0.040,Y -310.316,Z 1911.621,A 0.000,B 0.000,C 90.000,E1 291.770} C_DIS
LIN {X 0.169,Y -317.058,Z 1911.617,A 0.000,B 0.000,C 90.000,E1 290.972} C_DIS
LIN {X -0.107,Y -324.457,Z 1911.611,A 0.000,B 0.000,C 90.000,E1 290.066} C_DIS
LIN {X 0.039,Y -331.096,Z 1911.606,A 0.000,B 0.000,C 90.000,E1 289.087} C_DIS
LIN {X -0.166,Y -337.165,Z 1911.601,A 0.000,B 0.000,C 90.000,E1 288.181} C_DIS
LIN {X 0.001,Y -342.571,Z 1911.596,A 0.000,B 0.000,C 90.000,E1 287.221} C_DIS
LIN {X -0.103,Y -347.311,Z 1911.591,A 0.000,B 0.000,C 90.000,E1 286.315} C_DIS
LIN {X 0.070,Y -351.307,Z 1911.585,A 0.000,B 0.000,C 90.000,E1 285.371} C_DIS
LIN {X -0.050,Y -354.721,Z 1911.580,A 0.000,B 0.000,C 90.000,E1 284.481} C_DIS
LIN {X -0.028,Y -355.735,Z 1911.579,A 0.000,B 0.000,C 90.000,E1 284.175} C_DIS
LIN {X -0.143,Y -357.420,Z 1911.575,A 0.000,B 0.000,C 90.000,E1 283.592} C_DIS
LIN {X 0.098,Y -358.812,Z 1911.572,A 0.000,B 0.000,C 90.000,E1 282.952} C_DIS
LIN {X 0.081,Y -359.782,Z 1911.569,A 0.000,B 0.000,C 90.000,E1 282.355} C_DIS
LIN {X -0.007,Y -360.363,Z 1911.565,A 0.000,B 0.000,C 90.000,E1 281.771} C_DIS
LIN {X -0.089,Y -360.486,Z 1911.562,A 0.000,B 0.000,C 90.000,E1 281.186} C_DIS
LIN {X -0.167,Y -360.243,Z 1911.559,A 0.000,B 0.000,C 90.000,E1 280.602} C_DIS
LIN {X 0.109,Y -359.579,Z 1911.555,A 0.000,B 0.000,C 90.000,E1 279.962} C_DIS
LIN {X 0.028,Y -358.582,Z 1911.552,A 0.000,B 0.000,C 90.000,E1 279.378} C_DIS
LIN {X -0.113,Y -357.247,Z 1911.549,A 0.000,B 0.000,C 90.000,E1 278.803} C_DIS
LIN {X 0.147,Y -355.496,Z 1911.546,A 0.000,B 0.000,C 90.000,E1 278.163} C_DIS
LIN {X -0.061,Y -352.182,Z 1911.541,A 0.000,B 0.000,C 90.000,E1 277.296} C_DIS
LIN {X 0.119,Y -349.375,Z 1911.537,A 0.000,B 0.000,C 90.000,E1 276.663} C_DIS
LIN {X -0.065,Y -346.056,Z 1911.534,A 0.000,B 0.000,C 90.000,E1 276.087} C_DIS
LIN {X 0.079,Y -342.041,Z 1911.530,A 0.000,B 0.000,C 90.000,E1 275.454} C_DIS
LIN {X -0.140,Y -337.147,Z 1911.527,A 0.000,B 0.000,C 90.000,E1 274.878} C_DIS
LIN {X 0.027,Y -331.411,Z 1911.524,A 0.000,B 0.000,C 90.000,E1 274.245} C_DIS
LIN {X 0.157,Y -325.012,Z 1911.521,A 0.000,B 0.000,C 90.000,E1 273.669} C_DIS
LIN {X 0.070,Y -318.181,Z 1911.518,A 0.000,B 0.000,C 90.000,E1 273.212} C_DIS
LIN {X 0.139,Y -310.835,Z 1911.516,A 0.000,B 0.000,C 90.000,E1 272.808} C_DIS
LIN {X 0.054,Y -304.143,Z 1911.514,A 0.000,B 0.000,C 90.000,E1 272.579} C_DIS
LIN {X -0.149,Y -300.178,Z 1911.514,A 0.000,B 0.000,C 90.000,E1 272.522} C_DIS
LIN {X 0.094,Y -294.429,Z 1911.513,A 0.000,B 0.000,C 90.000,E1 272.407} C_DIS
LIN {X 0.027,Y -181.199,Z 1911.513,A 0.000,B 0.000,C 90.000,E1 272.407} C_DIS
LIN {X -0.049,Y -181.577,Z 1911.502,A 0.000,B 0.000,C 90.000,E1 270.401} C_DIS
LIN {X -0.072,Y -180.905,Z 1911.474,A 0.000,B 0.000,C 90.000,E1 265.355} C_DIS
LIN {X 0.002,Y -180.670,Z 1911.469,A 0.000,B 0.000,C 90.000,E1 264.489} C_DIS
LIN {X 0.076,Y -178.751,Z 1911.441,A 0.000,B 0.000,C 90.000,E1 259.398} C_DIS
LIN {X -0.026,Y -175.798,Z 1911.413,A 0.000,B 0.000,C 90.000,E1 254.338} C_DIS
LIN {X -0.031,Y -171.984,Z 1911.384,A 0.000,B 0.000,C 90.000,E1 249.209} C_DIS
LIN {X 0.007,Y -171.391,Z 1911.380,A 0.000,B 0.000,C 90.000,E1 248.337} C_DIS
LIN {X -0.008,Y -167.634,Z 1911.356,A 0.000,B 0.000,C 90.000,E1 244.024} C_DIS
LIN {X 0.006,Y -166.291,Z 1911.346,A 0.000,B 0.000,C 90.000,E1 242.281} C_DIS
LIN {X 0.001,Y -163.037,Z 1911.327,A 0.000,B 0.000,C 90.000,E1 238.791} C_DIS
LIN {X -0.037,Y -160.968,Z 1911.312,A 0.000,B 0.000,C 90.000,E1 236.167} C_DIS
LIN {X -0.060,Y -157.721,Z 1911.292,A 0.000,B 0.000,C 90.000,E1 232.637} C_DIS
LIN {X 0.099,Y -155.761,Z 1911.277,A 0.000,B 0.000,C 90.000,E1 229.908} C_DIS
LIN {X -0.064,Y -152.016,Z 1911.253,A 0.000,B 0.000,C 90.000,E1 225.486} C_DIS
LIN {X -0.046,Y -150.263,Z 1911.238,A 0.000,B 0.000,C 90.000,E1 222.771} C_DIS
LIN {X -0.028,Y -147.017,Z 1911.212,A 0.000,B 0.000,C 90.000,E1 218.222} C_DIS
LIN {X -0.007,Y -145.600,Z 1911.197,A 0.000,B 0.000,C 90.000,E1 215.471} C_DIS
LIN {X -0.003,Y -142.986,Z 1911.172,A 0.000,B 0.000,C 90.000,E1 210.875} C_DIS
LIN {X -0.003,Y -141.613,Z 1911.151,A 0.000,B 0.000,C 90.000,E1 207.180} C_DIS
LIN {X 0.039,Y -139.428,Z 1911.115,A 0.000,B 0.000,C 90.000,E1 200.663} C_DIS
LIN {X -0.043,Y -139.158,Z 1911.104,A 0.000,B 0.000,C 90.000,E1 198.833} C_DIS
LIN {X -0.025,Y -138.342,Z 1911.058,A 0.000,B 0.000,C 90.000,E1 190.423} C_DIS
LIN {X -0.043,Y -139.481,Z 1911.006,A 0.000,B 0.000,C 90.000,E1 181.088} C_DIS
LIN {X 0.038,Y -141.073,Z 1910.975,A 0.000,B 0.000,C 90.000,E1 175.469} C_DIS
LIN {X -0.008,Y -142.448,Z 1910.959,A 0.000,B 0.000,C 90.000,E1 172.704} C_DIS
LIN {X 0.082,Y -144.689,Z 1910.934,A 0.000,B 0.000,C 90.000,E1 168.049} C_DIS
LIN {X 0.035,Y -147.281,Z 1910.913,A 0.000,B 0.000,C 90.000,E1 164.393} C_DIS
LIN {X 0.051,Y -150.600,Z 1910.888,A 0.000,B 0.000,C 90.000,E1 159.826} C_DIS
LIN {X -0.013,Y -154.072,Z 1910.868,A 0.000,B 0.000,C 90.000,E1 156.230} C_DIS
LIN {X 0.053,Y -157.493,Z 1910.848,A 0.000,B 0.000,C 90.000,E1 152.615} C_DIS
LIN {X -0.001,Y -161.720,Z 1910.828,A 0.000,B 0.000,C 90.000,E1 149.076} C_DIS
LIN {X 0.013,Y -165.913,Z 1910.809,A 0.000,B 0.000,C 90.000,E1 145.548} C_DIS
LIN {X 0.000,Y -170.899,Z 1910.789,A 0.000,B 0.000,C 90.000,E1 142.065} C_DIS
LIN {X 0.026,Y -175.767,Z 1910.770,A 0.000,B 0.000,C 90.000,E1 138.609} C_DIS
LIN {X -0.101,Y -181.377,Z 1910.751,A 0.000,B 0.000,C 90.000,E1 135.243} C_DIS
LIN {X 0.032,Y -186.872,Z 1910.733,A 0.000,B 0.000,C 90.000,E1 131.838} C_DIS
LIN {X -0.016,Y -191.455,Z 1910.719,A 0.000,B 0.000,C 90.000,E1 129.358} C_DIS
LIN {X -0.083,Y -197.310,Z 1910.700,A 0.000,B 0.000,C 90.000,E1 126.091} C_DIS
LIN {X -0.048,Y -200.588,Z 1910.691,A 0.000,B 0.000,C 90.000,E1 124.452} C_DIS
LIN {X 0.029,Y -206.471,Z 1910.673,A 0.000,B 0.000,C 90.000,E1 121.209} C_DIS
LIN {X 0.021,Y -209.757,Z 1910.665,A 0.000,B 0.000,C 90.000,E1 119.617} C_DIS
LIN {X 0.053,Y -217.119,Z 1910.643,A 0.000,B 0.000,C 90.000,E1 115.668} C_DIS
LIN {X 0.008,Y -218.746,Z 1910.638,A 0.000,B 0.000,C 90.000,E1 114.899} C_DIS
LIN {X -0.088,Y -224.152,Z 1910.621,A 0.000,B 0.000,C 90.000,E1 111.844} C_DIS
LIN {X -0.141,Y -283.426,Z 1910.621,A 0.000,B 0.000,C 90.000,E1 111.844} C_DIS
LIN {X -0.045,Y -287.652,Z 1910.621,A 0.000,B 0.000,C 90.000,E1 111.716} C_DIS
LIN {X -0.143,Y -290.779,Z 1910.620,A 0.000,B 0.000,C 90.000,E1 111.535} C_DIS
LIN {X 0.096,Y -294.440,Z 1910.617,A 0.000,B 0.000,C 90.000,E1 111.099} C_DIS
LIN {X 0.145,Y -296.401,Z 1910.616,A 0.000,B 0.000,C 90.000,E1 110.791} C_DIS
LIN {X -0.049,Y -309.443,Z 1910.603,A 0.000,B 0.000,C 90.000,E1 108.544} C_DIS
LIN {X 0.056,Y -324.022,Z 1910.590,A 0.000,B 0.000,C 90.000,E1 106.260} C_DIS
LIN {X 0.112,Y -337.703,Z 1910.580,A 0.000,B 0.000,C 90.000,E1 104.356} C_DIS
LIN {X -0.070,Y -352.569,Z 1910.570,A 0.000,B 0.000,C 90.000,E1 102.535} C_DIS
LIN {X -0.056,Y -370.977,Z 1910.558,A 0.000,B 0.000,C 90.000,E1 100.489} C_DIS
LIN {X 0.021,Y -389.803,Z 1910.548,A 0.000,B 0.000,C 90.000,E1 98.624} C_DIS
LIN {X -0.079,Y -409.046,Z 1910.539,A 0.000,B 0.000,C 90.000,E1 96.947} C_DIS
LIN {X 0.164,Y -431.416,Z 1910.529,A 0.000,B 0.000,C 90.000,E1 95.163} C_DIS
LIN {X -0.103,Y -439.820,Z 1910.525,A 0.000,B 0.000,C 90.000,E1 94.588} C_DIS
LIN {X 0.114,Y -441.973,Z 1910.524,A 0.000,B 0.000,C 90.000,E1 94.359} C_DIS
LIN {X 0.011,Y -443.942,Z 1910.523,A 0.000,B 0.000,C 90.000,E1 94.131} C_DIS
LIN {X -0.061,Y -445.450,Z 1910.522,A 0.000,B 0.000,C 90.000,E1 93.898} C_DIS
LIN {X 0.120,Y -446.703,Z 1910.520,A 0.000,B 0.000,C 90.000,E1 93.612} C_DIS
LIN {X -0.144,Y -447.630,Z 1910.519,A 0.000,B 0.000,C 90.000,E1 93.383} C_DIS
LIN {X -0.185,Y -448.672,Z 1910.516,A 0.000,B 0.000,C 90.000,E1 92.865} C_DIS
LIN {X 0.205,Y -448.762,Z 1910.513,A 0.000,B 0.000,C 90.000,E1 92.293} C_DIS
LIN {X 0.170,Y -447.915,Z 1910.510,A 0.000,B 0.000,C 90.000,E1 91.776} C_DIS
LIN {X 0.120,Y -446.002,Z 1910.507,A 0.000,B 0.000,C 90.000,E1 91.260} C_DIS
LIN {X 0.067,Y -442.889,Z 1910.504,A 0.000,B 0.000,C 90.000,E1 90.745} C_DIS
LIN {X -0.046,Y -431.388,Z 1910.494,A 0.000,B 0.000,C 90.000,E1 88.912} C_DIS
LIN {X 0.047,Y -419.620,Z 1910.484,A 0.000,B 0.000,C 90.000,E1 87.020} C_DIS
LIN {X -0.055,Y -407.835,Z 1910.473,A 0.000,B 0.000,C 90.000,E1 85.122} C_DIS
LIN {X 0.015,Y -395.918,Z 1910.462,A 0.000,B 0.000,C 90.000,E1 83.166} C_DIS
LIN {X -0.033,Y -382.263,Z 1910.449,A 0.000,B 0.000,C 90.000,E1 80.905} C_DIS
LIN {X 0.036,Y -368.768,Z 1910.437,A 0.000,B 0.000,C 90.000,E1 78.578} C_DIS
LIN {X -0.171,Y -352.689,Z 1910.420,A 0.000,B 0.000,C 90.000,E1 75.644} C_DIS
LIN {X -0.154,Y -339.031,Z 1910.405,A 0.000,B 0.000,C 90.000,E1 72.906} C_DIS
LIN {X 0.143,Y -327.244,Z 1910.391,A 0.000,B 0.000,C 90.000,E1 70.369} C_DIS
LIN {X -0.001,Y -314.351,Z 1910.375,A 0.000,B 0.000,C 90.000,E1 67.539} C_DIS
LIN {X -0.141,Y -303.438,Z 1910.361,A 0.000,B 0.000,C 90.000,E1 64.973} C_DIS
LIN {X -0.035,Y -291.270,Z 1910.344,A 0.000,B 0.000,C 90.000,E1 61.975} C_DIS
LIN {X -0.018,Y -283.274,Z 1910.333,A 0.000,B 0.000,C 90.000,E1 59.950} C_DIS
LIN {X -0.105,Y -275.145,Z 1910.322,A 0.000,B 0.000,C 90.000,E1 57.916} C_DIS
LIN {X -0.037,Y -265.642,Z 1910.308,A 0.000,B 0.000,C 90.000,E1 55.468} C_DIS
LIN {X 0.048,Y -256.004,Z 1910.294,A 0.000,B 0.000,C 90.000,E1 52.970} C_DIS
LIN {X 0.079,Y -246.413,Z 1910.280,A 0.000,B 0.000,C 90.000,E1 50.436} C_DIS
LIN {X -0.024,Y -235.610,Z 1910.264,A 0.000,B 0.000,C 90.000,E1 47.514} C_DIS
LIN {X -0.066,Y -225.239,Z 1910.247,A 0.000,B 0.000,C 90.000,E1 44.514} C_DIS
LIN {X -0.048,Y -215.293,Z 1910.230,A 0.000,B 0.000,C 90.000,E1 41.434} C_DIS
LIN {X -0.077,Y -206.073,Z 1910.213,A 0.000,B 0.000,C 90.000,E1 38.302} C_DIS
LIN {X -0.072,Y -197.749,Z 1910.195,A 0.000,B 0.000,C 90.000,E1 35.105} C_DIS
LIN {X 0.105,Y -190.155,Z 1910.177,A 0.000,B 0.000,C 90.000,E1 31.799} C_DIS
LIN {X -0.047,Y -183.315,Z 1910.158,A 0.000,B 0.000,C 90.000,E1 28.537} C_DIS
LIN {X 0.024,Y -177.159,Z 1910.140,A 0.000,B 0.000,C 90.000,E1 25.155} C_DIS
LIN {X -0.038,Y -171.836,Z 1910.121,A 0.000,B 0.000,C 90.000,E1 21.770} C_DIS
LIN {X 0.001,Y -167.293,Z 1910.102,A 0.000,B 0.000,C 90.000,E1 18.308} C_DIS
LIN {X -0.012,Y -163.589,Z 1910.082,A 0.000,B 0.000,C 90.000,E1 14.828} C_DIS
LIN {X -0.020,Y -159.818,Z 1910.058,A 0.000,B 0.000,C 90.000,E1 10.433} C_DIS
LIN {X 0.064,Y -157.203,Z 1910.033,A 0.000,B 0.000,C 90.000,E1 5.967} C_DIS
LIN {X 0.000,Y -154.925,Z 1910.000,A 0.000,B 0.000,C 90.000,E1 360.000} C_DIS
LIN {X -0.010,Y -154.147,Z 1909.948,A 0.000,B 0.000,C 90.000,E1 350.557} C_DIS
LIN {X -0.004,Y -156.147,Z 1909.908,A 0.000,B 0.000,C 90.000,E1 343.378} C_DIS
LIN {X 0.029,Y -158.550,Z 1909.883,A 0.000,B 0.000,C 90.000,E1 338.901} C_DIS
LIN {X 0.043,Y -162.155,Z 1909.858,A 0.000,B 0.000,C 90.000,E1 334.460} C_DIS
LIN {X -0.051,Y -166.082,Z 1909.839,A 0.000,B 0.000,C 90.000,E1 330.973} C_DIS
LIN {X 0.048,Y -170.976,Z 1909.819,A 0.000,B 0.000,C 90.000,E1 327.454} C_DIS
LIN {X -0.041,Y -175.290,Z 1909.805,A 0.000,B 0.000,C 90.000,E1 324.895} C_DIS
LIN {X 0.013,Y -180.273,Z 1909.791,A 0.000,B 0.000,C 90.000,E1 322.316} C_DIS
LIN {X 0.013,Y -186.136,Z 1909.777,A 0.000,B 0.000,C 90.000,E1 319.784} C_DIS
LIN {X -0.020,Y -191.740,Z 1909.765,A 0.000,B 0.000,C 90.000,E1 317.715} C_DIS
LIN {X 0.018,Y -199.386,Z 1909.751,A 0.000,B 0.000,C 90.000,E1 315.243} C_DIS
LIN {X -0.080,Y -207.978,Z 1909.738,A 0.000,B 0.000,C 90.000,E1 312.852} C_DIS
LIN {X -0.099,Y -219.056,Z 1909.723,A 0.000,B 0.000,C 90.000,E1 310.092} C_DIS
LIN {X 0.024,Y -231.170,Z 1909.708,A 0.000,B 0.000,C 90.000,E1 307.363} C_DIS
LIN {X -0.156,Y -246.114,Z 1909.691,A 0.000,B 0.000,C 90.000,E1 304.405} C_DIS
LIN {X -0.151,Y -257.966,Z 1909.679,A 0.000,B 0.000,C 90.000,E1 302.212} C_DIS
LIN {X 0.091,Y -272.036,Z 1909.665,A 0.000,B 0.000,C 90.000,E1 299.667} C_DIS
LIN {X -0.135,Y -281.927,Z 1909.655,A 0.000,B 0.000,C 90.000,E1 297.975} C_DIS
LIN {X 0.039,Y -291.529,Z 1909.646,A 0.000,B 0.000,C 90.000,E1 296.232} C_DIS
LIN {X 0.121,Y -296.974,Z 1909.640,A 0.000,B 0.000,C 90.000,E1 295.207} C_DIS
LIN {X 0.124,Y -301.786,Z 1909.635,A 0.000,B 0.000,C 90.000,E1 294.207} C_DIS
LIN {X 0.010,Y -304.577,Z 1909.631,A 0.000,B 0.000,C 90.000,E1 293.567} C_DIS
LIN {X -0.030,Y -308.047,Z 1909.625,A 0.000,B 0.000,C 90.000,E1 292.589} C_DIS
LIN {X -0.057,Y -308.460,Z 1909.625,A 0.000,B 0.000,C 90.000,E1 292.461} C_DIS
LIN {X -0.112,Y -308.507,Z 1909.625,A 0.000,B 0.000,C 90.000,E1 292.461} C_DIS
LIN {X 0.136,Y -315.287,Z 1909.620,A 0.000,B 0.000,C 90.000,E1 291.589} C_DIS
LIN {X -0.098,Y -322.550,Z 1909.615,A 0.000,B 0.000,C 90.000,E1 290.663} C_DIS
LIN {X 0.028,Y -329.125,Z 1909.609,A 0.000,B 0.000,C 90.000,E1 289.685} C_DIS
LIN {X 0.120,Y -335.125,Z 1909.604,A 0.000,B 0.000,C 90.000,E1 288.725} C_DIS
LIN {X -0.054,Y -340.668,Z 1909.599,A 0.000,B 0.000,C 90.000,E1 287.819} C_DIS
LIN {X 0.155,Y -345.575,Z 1909.594,A 0.000,B 0.000,C 90.000,E1 286.858} C_DIS
LIN {X -0.023,Y -349.832,Z 1909.589,A 0.000,B 0.000,C 90.000,E1 285.969} C_DIS
LIN {X -0.063,Y -353.508,Z 1909.584,A 0.000,B 0.000,C 90.000,E1 285.064} C_DIS
LIN {X 0.175,Y -356.584,Z 1909.579,A 0.000,B 0.000,C 90.000,E1 284.120} C_DIS
LIN {X 0.058,Y -358.197,Z 1909.575,A 0.000,B 0.000,C 90.000,E1 283.536} C_DIS
LIN {X 0.038,Y -359.524,Z 1909.572,A 0.000,B 0.000,C 90.000,E1 282.939} C_DIS
LIN {X -0.055,Y -360.451,Z 1909.569,A 0.000,B 0.000,C 90.000,E1 282.355} C_DIS
LIN {X -0.139,Y -360.998,Z 1909.565,A 0.000,B 0.000,C 90.000,E1 281.771} C_DIS
LIN {X 0.137,Y -361.115,Z 1909.562,A 0.000,B 0.000,C 90.000,E1 281.130} C_DIS
LIN {X 0.063,Y -360.846,Z 1909.559,A 0.000,B 0.000,C 90.000,E1 280.546} C_DIS
LIN {X -0.011,Y -360.185,Z 1909.555,A 0.000,B 0.000,C 90.000,E1 279.962} C_DIS
LIN {X -0.088,Y -359.195,Z 1909.552,A 0.000,B 0.000,C 90.000,E1 279.378} C_DIS
LIN {X 0.128,Y -357.882,Z 1909.549,A 0.000,B 0.000,C 90.000,E1 278.746} C_DIS
LIN {X 0.039,Y -356.169,Z 1909.545,A 0.000,B 0.000,C 90.000,E1 278.163} C_DIS
LIN {X -0.162,Y -352.933,Z 1909.540,A 0.000,B 0.000,C 90.000,E1 277.296} C_DIS
LIN {X 0.023,Y -350.212,Z 1909.537,A 0.000,B 0.000,C 90.000,E1 276.663} C_DIS
LIN {X -0.155,Y -347.026,Z 1909.534,A 0.000,B 0.000,C 90.000,E1 276.087} C_DIS
LIN {X -0.004,Y -343.197,Z 1909.530,A 0.000,B 0.000,C 90.000,E1 275.454} C_DIS
LIN {X 0.121,Y -338.566,Z 1909.527,A 0.000,B 0.000,C 90.000,E1 274.821} C_DIS
LIN {X -0.115,Y -333.100,Z 1909.523,A 0.000,B 0.000,C 90.000,E1 274.245} C_DIS
LIN {X -0.152,Y -326.889,Z 1909.520,A 0.000,B 0.000,C 90.000,E1 273.669} C_DIS
LIN {X -0.077,Y -323.595,Z 1909.519,A 0.000,B 0.000,C 90.000,E1 273.383} C_DIS
LIN {X 0.135,Y -316.646,Z 1909.516,A 0.000,B 0.000,C 90.000,E1 272.865} C_DIS
LIN {X 0.152,Y -309.311,Z 1909.514,A 0.000,B 0.000,C 90.000,E1 272.465} C_DIS
LIN {X -0.063,Y -305.661,Z 1909.513,A 0.000,B 0.000,C 90.000,E1 272.350} C_DIS
LIN {X 0.002,Y -298.511,Z 1909.512,A 0.000,B 0.000,C 90.000,E1 272.121} C_DIS
LIN {X 0.127,Y -293.313,Z 1909.511,A 0.000,B 0.000,C 90.000,E1 272.007} C_DIS
LIN {X 0.053,Y -291.372,Z 1909.511,A 0.000,B 0.000,C 90.000,E1 272.007} C_DIS
LIN {X 0.010,Y -181.261,Z 1909.511,A 0.000,B 0.000,C 90.000,E1 272.007} C_DIS
LIN {X 0.009,Y -181.581,Z 1909.502,A 0.000,B 0.000,C 90.000,E1 270.286} C_DIS
LIN {X -0.015,Y -180.899,Z 1909.474,A 0.000,B 0.000,C 90.000,E1 265.241} C_DIS
LIN {X -0.066,Y -180.216,Z 1909.464,A 0.000,B 0.000,C 90.000,E1 263.571} C_DIS
LIN {X 0.064,Y -179.034,Z 1909.445,A 0.000,B 0.000,C 90.000,E1 260.151} C_DIS
LIN {X -0.049,Y -178.692,Z 1909.441,A 0.000,B 0.000,C 90.000,E1 259.342} C_DIS
LIN {X 0.062,Y -175.741,Z 1909.412,A 0.000,B 0.000,C 90.000,E1 254.212} C_DIS
LIN {X 0.056,Y -171.925,Z 1909.384,A 0.000,B 0.000,C 90.000,E1 249.082} C_DIS
LIN {X 0.031,Y -171.299,Z 1909.379,A 0.000,B 0.000,C 90.000,E1 248.230} C_DIS
LIN {X 0.076,Y -167.561,Z 1909.355,A 0.000,B 0.000,C 90.000,E1 243.896} C_DIS
LIN {X 0.090,Y -166.187,Z 1909.345,A 0.000,B 0.000,C 90.000,E1 242.153} C_DIS
LIN {X 0.079,Y -162.957,Z 1909.326,A 0.000,B 0.000,C 90.000,E1 238.663} C_DIS
LIN {X -0.097,Y -160.865,Z 1909.311,A 0.000,B 0.000,C 90.000,E1 236.087} C_DIS
LIN {X 0.008,Y -157.639,Z 1909.292,A 0.000,B 0.000,C 90.000,E1 232.512} C_DIS
LIN {X 0.041,Y -155.677,Z 1909.277,A 0.000,B 0.000,C 90.000,E1 229.828} C_DIS
LIN {X -0.015,Y -151.943,Z 1909.252,A 0.000,B 0.000,C 90.000,E1 225.364} C_DIS
LIN {X -0.003,Y -150.182,Z 1909.237,A 0.000,B 0.000,C 90.000,E1 222.651} C_DIS
LIN {X 0.027,Y -146.955,Z 1909.212,A 0.000,B 0.000,C 90.000,E1 218.096} C_DIS
LIN {X -0.070,Y -145.543,Z 1909.196,A 0.000,B 0.000,C 90.000,E1 215.391} C_DIS
LIN {X -0.069,Y -142.938,Z 1909.171,A 0.000,B 0.000,C 90.000,E1 210.797} C_DIS
LIN {X -0.012,Y -141.562,Z 1909.150,A 0.000,B 0.000,C 90.000,E1 207.078} C_DIS
LIN {X 0.041,Y -139.410,Z 1909.114,A 0.000,B 0.000,C 90.000,E1 200.556} C_DIS
LIN {X -0.037,Y -139.131,Z 1909.104,A 0.000,B 0.000,C 90.000,E1 198.725} C_DIS
LIN {X -0.011,Y -138.350,Z 1909.057,A 0.000,B 0.000,C 90.000,E1 190.310} C_DIS
LIN {X -0.023,Y -139.498,Z 1909.005,A 0.000,B 0.000,C 90.000,E1 180.974} C_DIS
LIN {X 0.057,Y -141.118,Z 1908.974,A 0.000,B 0.000,C 90.000,E1 175.355} C_DIS
LIN {X 0.011,Y -142.497,Z 1908.959,A 0.000,B 0.000,C 90.000,E1 172.591} C_DIS
LIN {X -0.042,Y -144.752,Z 1908.933,A 0.000,B 0.000,C 90.000,E1 167.993} C_DIS
LIN {X 0.050,Y -147.361,Z 1908.913,A 0.000,B 0.000,C 90.000,E1 164.283} C_DIS
LIN {X -0.028,Y -150.688,Z 1908.887,A 0.000,B 0.000,C 90.000,E1 159.752} C_DIS
LIN {X 0.055,Y -154.168,Z 1908.867,A 0.000,B 0.000,C 90.000,E1 156.102} C_DIS
LIN {X -0.015,Y -157.601,Z 1908.847,A 0.000,B 0.000,C 90.000,E1 152.538} C_DIS
LIN {X -0.065,Y -161.853,Z 1908.828,A 0.000,B 0.000,C 90.000,E1 148.997} C_DIS
LIN {X -0.047,Y -166.043,Z 1908.808,A 0.000,B 0.000,C 90.000,E1 145.468} C_DIS
LIN {X -0.056,Y -171.047,Z 1908.789,A 0.000,B 0.000,C 90.000,E1 141.984} C_DIS
LIN {X -0.025,Y -175.919,Z 1908.770,A 0.000,B 0.000,C 90.000,E1 138.528} C_DIS
LIN {X -0.034,Y -180.157,Z 1908.755,A 0.000,B 0.000,C 90.000,E1 135.972} C_DIS
LIN {X -0.065,Y -185.575,Z 1908.737,A 0.000,B 0.000,C 90.000,E1 132.609} C_DIS
LIN {X -0.015,Y -190.163,Z 1908.723,A 0.000,B 0.000,C 90.000,E1 130.092} C_DIS
LIN {X 0.031,Y -197.492,Z 1908.700,A 0.000,B 0.000,C 90.000,E1 125.964} C_DIS
LIN {X 0.073,Y -200.762,Z 1908.691,A 0.000,B 0.000,C 90.000,E1 124.326} C_DIS
LIN {X -0.016,Y -206.653,Z 1908.673,A 0.000,B 0.000,C 90.000,E1 121.131} C_DIS
LIN {X -0.025,Y -209.948,Z 1908.664,A 0.000,B 0.000,C 90.000,E1 119.539} C_DIS
LIN {X 0.003,Y -217.302,Z 1908.642,A 0.000,B 0.000,C 90.000,E1 115.591} C_DIS
LIN {X -0.042,Y -218.926,Z 1908.638,A 0.000,B 0.000,C 90.000,E1 114.823} C_DIS
LIN {X -0.071,Y -224.145,Z 1908.621,A 0.000,B 0.000,C 90.000,E1 111.844} C_DIS
LIN {X -0.128,Y -283.030,Z 1908.621,A 0.000,B 0.000,C 90.000,E1 111.844} C_DIS
LIN {X 0.057,Y -284.740,Z 1908.621,A 0.000,B 0.000,C 90.000,E1 111.791} C_DIS
LIN {X -0.006,Y -287.510,Z 1908.621,A 0.000,B 0.000,C 90.000,E1 111.716} C_DIS
LIN {X -0.103,Y -290.695,Z 1908.620,A 0.000,B 0.000,C 90.000,E1 111.535} C_DIS
LIN {X -0.107,Y -294.338,Z 1908.617,A 0.000,B 0.000,C 90.000,E1 111.153} C_DIS
LIN {X 0.057,Y -299.768,Z 1908.612,A 0.000,B 0.000,C 90.000,E1 110.194} C_DIS
LIN {X 0.133,Y -313.362,Z 1908.599,A 0.000,B 0.000,C 90.000,E1 107.873} C_DIS
LIN {X -0.074,Y -328.343,Z 1908.587,A 0.000,B 0.000,C 90.000,E1 105.662} C_DIS
LIN {X -0.025,Y -342.399,Z 1908.577,A 0.000,B 0.000,C 90.000,E1 103.772} C_DIS
LIN {X -0.092,Y -357.634,Z 1908.566,A 0.000,B 0.000,C 90.000,E1 101.951} C_DIS
LIN {X -0.101,Y -376.184,Z 1908.555,A 0.000,B 0.000,C 90.000,E1 99.962} C_DIS
LIN {X -0.149,Y -395.122,Z 1908.545,A 0.000,B 0.000,C 90.000,E1 98.163} C_DIS
LIN {X 0.095,Y -417.229,Z 1908.535,A 0.000,B 0.000,C 90.000,E1 96.258} C_DIS
LIN {X -0.026,Y -439.692,Z 1908.526,A 0.000,B 0.000,C 90.000,E1 94.588} C_DIS
LIN {X 0.190,Y -441.875,Z 1908.524,A 0.000,B 0.000,C 90.000,E1 94.359} C_DIS
LIN {X 0.103,Y -443.849,Z 1908.523,A 0.000,B 0.000,C 90.000,E1 94.131} C_DIS
LIN {X 0.048,Y -445.364,Z 1908.522,A 0.000,B 0.000,C 90.000,E1 93.898} C_DIS
LIN {X -0.218,Y -446.635,Z 1908.520,A 0.000,B 0.000,C 90.000,E1 93.669} C_DIS
LIN {X -0.036,Y -447.577,Z 1908.519,A 0.000,B 0.000,C 90.000,E1 93.383} C_DIS
LIN {X -0.077,Y -448.644,Z 1908.516,A 0.000,B 0.000,C 90.000,E1 92.865} C_DIS
LIN {X -0.135,Y -448.757,Z 1908.513,A 0.000,B 0.000,C 90.000,E1 92.350} C_DIS
LIN {X -0.169,Y -447.935,Z 1908.510,A 0.000,B 0.000,C 90.000,E1 91.833} C_DIS
LIN {X -0.219,Y -446.051,Z 1908.507,A 0.000,B 0.000,C 90.000,E1 91.318} C_DIS
LIN {X 0.174,Y -442.956,Z 1908.504,A 0.000,B 0.000,C 90.000,E1 90.745} C_DIS
LIN {X 0.059,Y -431.454,Z 1908.494,A 0.000,B 0.000,C 90.000,E1 88.912} C_DIS
LIN {X 0.150,Y -419.691,Z 1908.484,A 0.000,B 0.000,C 90.000,E1 87.020} C_DIS
LIN {X 0.047,Y -407.904,Z 1908.473,A 0.000,B 0.000,C 90.000,E1 85.122} C_DIS
LIN {X 0.116,Y -395.988,Z 1908.462,A 0.000,B 0.000,C 90.000,E1 83.166} C_DIS
LIN {X 0.067,Y -382.333,Z 1908.450,A 0.000,B 0.000,C 90.000,E1 80.905} C_DIS
LIN {X 0.132,Y -368.835,Z 1908.437,A 0.000,B 0.000,C 90.000,E1 78.578} C_DIS
LIN {X -0.076,Y -352.749,Z 1908.420,A 0.000,B 0.000,C 90.000,E1 75.644} C_DIS
LIN {X -0.062,Y -339.089,Z 1908.405,A 0.000,B 0.000,C 90.000,E1 72.906} C_DIS
LIN {X -0.074,Y -327.299,Z 1908.391,A 0.000,B 0.000,C 90.000,E1 70.423} C_DIS
LIN {X 0.088,Y -314.404,Z 1908.375,A 0.000,B 0.000,C 90.000,E1 67.539} C_DIS
LIN {X -0.055,Y -303.485,Z 1908.361,A 0.000,B 0.000,C 90.000,E1 64.973} C_DIS
LIN {X 0.055,Y -292.632,Z 1908.346,A 0.000,B 0.000,C 90.000,E1 62.308} C_DIS
LIN {X -0.154,Y -284.667,Z 1908.335,A 0.000,B 0.000,C 90.000,E1 60.333} C_DIS
LIN {X 0.027,Y -276.555,Z 1908.324,A 0.000,B 0.000,C 90.000,E1 58.250} C_DIS
LIN {X 0.120,Y -267.057,Z 1908.310,A 0.000,B 0.000,C 90.000,E1 55.801} C_DIS
LIN {X 0.085,Y -257.424,Z 1908.296,A 0.000,B 0.000,C 90.000,E1 53.336} C_DIS
LIN {X 0.141,Y -247.833,Z 1908.282,A 0.000,B 0.000,C 90.000,E1 50.803} C_DIS
LIN {X -0.089,Y -236.990,Z 1908.266,A 0.000,B 0.000,C 90.000,E1 47.919} C_DIS
LIN {X -0.095,Y -226.546,Z 1908.249,A 0.000,B 0.000,C 90.000,E1 44.919} C_DIS
LIN {X 0.021,Y -215.334,Z 1908.230,A 0.000,B 0.000,C 90.000,E1 41.434} C_DIS
LIN {X -0.010,Y -206.110,Z 1908.213,A 0.000,B 0.000,C 90.000,E1 38.302} C_DIS
LIN {X -0.007,Y -197.785,Z 1908.195,A 0.000,B 0.000,C 90.000,E1 35.105} C_DIS
LIN {X -0.092,Y -190.188,Z 1908.177,A 0.000,B 0.000,C 90.000,E1 31.878} C_DIS
LIN {X -0.072,Y -183.346,Z 1908.159,A 0.000,B 0.000,C 90.000,E1 28.565} C_DIS
LIN {X -0.074,Y -177.186,Z 1908.140,A 0.000,B 0.000,C 90.000,E1 25.207} C_DIS
LIN {X 0.022,Y -171.858,Z 1908.121,A 0.000,B 0.000,C 90.000,E1 21.770} C_DIS
LIN {X 0.060,Y -167.312,Z 1908.102,A 0.000,B 0.000,C 90.000,E1 18.308} C_DIS
LIN {X 0.046,Y -163.601,Z 1908.083,A 0.000,B 0.000,C 90.000,E1 14.828} C_DIS
LIN {X 0.038,Y -159.825,Z 1908.058,A 0.000,B 0.000,C 90.000,E1 10.433} C_DIS
LIN {X -0.036,Y -157.206,Z 1908.033,A 0.000,B 0.000,C 90.000,E1 6.024} C_DIS
LIN {X 0.000,Y -154.917,Z 1908.000,A 0.000,B 0.000,C 90.000,E1 360.000} C_DIS
LIN {X -0.010,Y -154.140,Z 1907.948,A 0.000,B 0.000,C 90.000,E1 350.557} C_DIS
LIN {X -0.005,Y -156.141,Z 1907.908,A 0.000,B 0.000,C 90.000,E1 343.378} C_DIS
LIN {X 0.028,Y -158.547,Z 1907.883,A 0.000,B 0.000,C 90.000,E1 338.901} C_DIS
LIN {X 0.042,Y -162.155,Z 1907.858,A 0.000,B 0.000,C 90.000,E1 334.460} C_DIS
LIN {X -0.051,Y -166.084,Z 1907.839,A 0.000,B 0.000,C 90.000,E1 330.973} C_DIS
LIN {X 0.046,Y -170.981,Z 1907.819,A 0.000,B 0.000,C 90.000,E1 327.454} C_DIS
LIN {X -0.042,Y -175.297,Z 1907.805,A 0.000,B 0.000,C 90.000,E1 324.895} C_DIS
LIN {X 0.012,Y -180.281,Z 1907.791,A 0.000,B 0.000,C 90.000,E1 322.316} C_DIS
LIN {X 0.012,Y -186.144,Z 1907.777,A 0.000,B 0.000,C 90.000,E1 319.784} C_DIS
LIN {X -0.021,Y -191.748,Z 1907.765,A 0.000,B 0.000,C 90.000,E1 317.715} C_DIS
LIN {X 0.017,Y -199.393,Z 1907.751,A 0.000,B 0.000,C 90.000,E1 315.243} C_DIS
LIN {X -0.080,Y -207.985,Z 1907.738,A 0.000,B 0.000,C 90.000,E1 312.852} C_DIS
LIN {X -0.099,Y -219.064,Z 1907.723,A 0.000,B 0.000,C 90.000,E1 310.092} C_DIS
LIN {X 0.024,Y -231.179,Z 1907.708,A 0.000,B 0.000,C 90.000,E1 307.363} C_DIS
LIN {X -0.157,Y -246.125,Z 1907.691,A 0.000,B 0.000,C 90.000,E1 304.405} C_DIS
LIN {X -0.151,Y -257.976,Z 1907.679,A 0.000,B 0.000,C 90.000,E1 302.212} C_DIS
LIN {X 0.092,Y -272.044,Z 1907.665,A 0.000,B 0.000,C 90.000,E1 299.667} C_DIS
LIN {X -0.133,Y -281.935,Z 1907.655,A 0.000,B 0.000,C 90.000,E1 297.975} C_DIS
LIN {X 0.040,Y -291.539,Z 1907.646,A 0.000,B 0.000,C 90.000,E1 296.232} C_DIS
LIN {X 0.122,Y -296.986,Z 1907.640,A 0.000,B 0.000,C 90.000,E1 295.207} C_DIS
LIN {X 0.125,Y -301.796,Z 1907.635,A 0.000,B 0.000,C 90.000,E1 294.207} C_DIS
LIN {X 0.012,Y -304.586,Z 1907.631,A 0.000,B 0.000,C 90.000,E1 293.567} C_DIS
LIN {X 0.041,Y -306.400,Z 1907.628,A 0.000,B 0.000,C 90.000,E1 293.078} C_DIS
LIN {X -0.014,Y -306.453,Z 1907.628,A 0.000,B 0.000,C 90.000,E1 293.078} C_DIS
LIN {X -0.099,Y -315.300,Z 1907.622,A 0.000,B 0.000,C 90.000,E1 291.950} C_DIS
LIN {X -0.046,Y -322.275,Z 1907.616,A 0.000,B 0.000,C 90.000,E1 290.972} C_DIS
LIN {X 0.087,Y -328.653,Z 1907.611,A 0.000,B 0.000,C 90.000,E1 289.993} C_DIS
LIN {X 0.144,Y -336.350,Z 1907.604,A 0.000,B 0.000,C 90.000,E1 288.725} C_DIS
LIN {X -0.017,Y -341.661,Z 1907.599,A 0.000,B 0.000,C 90.000,E1 287.819} C_DIS
LIN {X -0.129,Y -346.381,Z 1907.594,A 0.000,B 0.000,C 90.000,E1 286.913} C_DIS
LIN {X 0.033,Y -350.524,Z 1907.589,A 0.000,B 0.000,C 90.000,E1 285.969} C_DIS
LIN {X -0.001,Y -354.128,Z 1907.584,A 0.000,B 0.000,C 90.000,E1 285.064} C_DIS
LIN {X -0.102,Y -357.189,Z 1907.579,A 0.000,B 0.000,C 90.000,E1 284.175} C_DIS
LIN {X 0.132,Y -358.815,Z 1907.575,A 0.000,B 0.000,C 90.000,E1 283.536} C_DIS
LIN {X 0.115,Y -360.108,Z 1907.572,A 0.000,B 0.000,C 90.000,E1 282.939} C_DIS
LIN {X 0.026,Y -360.979,Z 1907.569,A 0.000,B 0.000,C 90.000,E1 282.355} C_DIS
LIN {X -0.055,Y -361.489,Z 1907.565,A 0.000,B 0.000,C 90.000,E1 281.771} C_DIS
LIN {X -0.130,Y -361.634,Z 1907.562,A 0.000,B 0.000,C 90.000,E1 281.186} C_DIS
LIN {X 0.154,Y -361.344,Z 1907.559,A 0.000,B 0.000,C 90.000,E1 280.546} C_DIS
LIN {X 0.083,Y -360.676,Z 1907.555,A 0.000,B 0.000,C 90.000,E1 279.962} C_DIS
LIN {X 0.009,Y -359.664,Z 1907.552,A 0.000,B 0.000,C 90.000,E1 279.378} C_DIS
LIN {X -0.127,Y -358.363,Z 1907.549,A 0.000,B 0.000,C 90.000,E1 278.803} C_DIS
LIN {X 0.141,Y -356.689,Z 1907.546,A 0.000,B 0.000,C 90.000,E1 278.163} C_DIS
LIN {X -0.057,Y -353.530,Z 1907.541,A 0.000,B 0.000,C 90.000,E1 277.296} C_DIS
LIN {X 0.132,Y -350.897,Z 1907.537,A 0.000,B 0.000,C 90.000,E1 276.663} C_DIS
LIN {X -0.044,Y -347.841,Z 1907.534,A 0.000,B 0.000,C 90.000,E1 276.087} C_DIS
LIN {X 0.110,Y -344.161,Z 1907.530,A 0.000,B 0.000,C 90.000,E1 275.454} C_DIS
LIN {X -0.099,Y -339.763,Z 1907.527,A 0.000,B 0.000,C 90.000,E1 274.878} C_DIS
LIN {X 0.007,Y -334.582,Z 1907.524,A 0.000,B 0.000,C 90.000,E1 274.245} C_DIS
LIN {X -0.110,Y -328.671,Z 1907.520,A 0.000,B 0.000,C 90.000,E1 273.669} C_DIS
LIN {X 0.067,Y -322.311,Z 1907.517,A 0.000,B 0.000,C 90.000,E1 273.094} C_DIS
LIN {X -0.032,Y -315.514,Z 1907.515,A 0.000,B 0.000,C 90.000,E1 272.636} C_DIS
LIN {X -0.031,Y -308.336,Z 1907.512,A 0.000,B 0.000,C 90.000,E1 272.236} C_DIS
LIN {X 0.095,Y -300.386,Z 1907.511,A 0.000,B 0.000,C 90.000,E1 271.892} C_DIS
LIN {X 0.004,Y -292.213,Z 1907.510,A 0.000,B 0.000,C 90.000,E1 271.718} C_DIS
LIN {X 0.064,Y -287.495,Z 1907.509,A 0.000,B 0.000,C 90.000,E1 271.661} C_DIS
LIN {X 0.011,Y -181.320,Z 1907.509,A 0.000,B 0.000,C 90.000,E1 271.661} C_DIS
LIN {X -0.085,Y -181.545,Z 1907.500,A 0.000,B 0.000,C 90.000,E1 269.943} C_DIS
LIN {X 0.081,Y -180.824,Z 1907.471,A 0.000,B 0.000,C 90.000,E1 264.837} C_DIS
LIN {X -0.020,Y -178.930,Z 1907.443,A 0.000,B 0.000,C 90.000,E1 259.803} C_DIS
LIN {X 0.018,Y -175.978,Z 1907.415,A 0.000,B 0.000,C 90.000,E1 254.700} C_DIS
LIN {X -0.036,Y -175.466,Z 1907.410,A 0.000,B 0.000,C 90.000,E1 253.866} C_DIS
LIN {X 0.021,Y -172.216,Z 1907.387,A 0.000,B 0.000,C 90.000,E1 249.571} C_DIS
LIN {X -0.002,Y -171.692,Z 1907.382,A 0.000,B 0.000,C 90.000,E1 248.720} C_DIS
LIN {X -0.011,Y -167.919,Z 1907.358,A 0.000,B 0.000,C 90.000,E1 244.409} C_DIS
LIN {X 0.007,Y -166.661,Z 1907.348,A 0.000,B 0.000,C 90.000,E1 242.666} C_DIS
LIN {X -0.078,Y -162.645,Z 1907.324,A 0.000,B 0.000,C 90.000,E1 238.329} C_DIS
LIN {X -0.016,Y -161.333,Z 1907.314,A 0.000,B 0.000,C 90.000,E1 236.548} C_DIS
LIN {X 0.028,Y -157.328,Z 1907.290,A 0.000,B 0.000,C 90.000,E1 232.110} C_DIS
LIN {X -0.039,Y -155.311,Z 1907.275,A 0.000,B 0.000,C 90.000,E1 229.461} C_DIS
LIN {X -0.001,Y -151.667,Z 1907.250,A 0.000,B 0.000,C 90.000,E1 224.960} C_DIS
LIN {X 0.043,Y -150.533,Z 1907.240,A 0.000,B 0.000,C 90.000,E1 223.137} C_DIS
LIN {X -0.026,Y -147.258,Z 1907.214,A 0.000,B 0.000,C 90.000,E1 218.624} C_DIS
LIN {X 0.030,Y -145.284,Z 1907.194,A 0.000,B 0.000,C 90.000,E1 214.945} C_DIS
LIN {X 0.063,Y -142.385,Z 1907.164,A 0.000,B 0.000,C 90.000,E1 209.411} C_DIS
LIN {X -0.014,Y -141.363,Z 1907.148,A 0.000,B 0.000,C 90.000,E1 206.668} C_DIS
LIN {X -0.036,Y -139.343,Z 1907.112,A 0.000,B 0.000,C 90.000,E1 200.174} C_DIS
LIN {X -0.030,Y -139.013,Z 1907.102,A 0.000,B 0.000,C 90.000,E1 198.308} C_DIS
LIN {X -0.034,Y -138.341,Z 1907.055,A 0.000,B 0.000,C 90.000,E1 189.905} C_DIS
LIN {X -0.015,Y -139.397,Z 1907.008,A 0.000,B 0.000,C 90.000,E1 181.489} C_DIS
LIN {X 0.039,Y -141.300,Z 1906.972,A 0.000,B 0.000,C 90.000,E1 174.951} C_DIS
LIN {X -0.004,Y -142.661,Z 1906.957,A 0.000,B 0.000,C 90.000,E1 172.186} C_DIS
LIN {X -0.054,Y -145.006,Z 1906.931,A 0.000,B 0.000,C 90.000,E1 167.589} C_DIS
LIN {X -0.064,Y -147.632,Z 1906.911,A 0.000,B 0.000,C 90.000,E1 163.921} C_DIS
LIN {X 0.013,Y -150.263,Z 1906.890,A 0.000,B 0.000,C 90.000,E1 160.242} C_DIS
LIN {X 0.027,Y -153.662,Z 1906.870,A 0.000,B 0.000,C 90.000,E1 156.613} C_DIS
LIN {X 0.083,Y -157.077,Z 1906.850,A 0.000,B 0.000,C 90.000,E1 152.999} C_DIS
LIN {X 0.022,Y -161.210,Z 1906.830,A 0.000,B 0.000,C 90.000,E1 149.459} C_DIS
LIN {X -0.030,Y -163.301,Z 1906.821,A 0.000,B 0.000,C 90.000,E1 147.709} C_DIS
LIN {X -0.020,Y -167.749,Z 1906.801,A 0.000,B 0.000,C 90.000,E1 144.196} C_DIS
LIN {X -0.002,Y -171.566,Z 1906.787,A 0.000,B 0.000,C 90.000,E1 141.582} C_DIS
LIN {X -0.068,Y -176.512,Z 1906.767,A 0.000,B 0.000,C 90.000,E1 138.162} C_DIS
LIN {X 0.057,Y -180.810,Z 1906.753,A 0.000,B 0.000,C 90.000,E1 135.567} C_DIS
LIN {X 0.042,Y -186.219,Z 1906.734,A 0.000,B 0.000,C 90.000,E1 132.204} C_DIS
LIN {X -0.019,Y -190.856,Z 1906.721,A 0.000,B 0.000,C 90.000,E1 129.725} C_DIS
LIN {X 0.015,Y -196.617,Z 1906.702,A 0.000,B 0.000,C 90.000,E1 126.423} C_DIS
LIN {X -0.073,Y -199.855,Z 1906.693,A 0.000,B 0.000,C 90.000,E1 124.818} C_DIS
LIN {X 0.123,Y -204.254,Z 1906.680,A 0.000,B 0.000,C 90.000,E1 122.339} C_DIS
LIN {X -0.093,Y -210.605,Z 1906.662,A 0.000,B 0.000,C 90.000,E1 119.205} C_DIS
LIN {X 0.002,Y -216.420,Z 1906.645,A 0.000,B 0.000,C 90.000,E1 116.027} C_DIS
LIN {X 0.013,Y -219.544,Z 1906.636,A 0.000,B 0.000,C 90.000,E1 114.463} C_DIS
LIN {X -0.078,Y -224.148,Z 1906.621,A 0.000,B 0.000,C 90.000,E1 111.844} C_DIS
LIN {X -0.128,Y -283.498,Z 1906.621,A 0.000,B 0.000,C 90.000,E1 111.844} C_DIS
LIN {X 0.036,Y -289.624,Z 1906.620,A 0.000,B 0.000,C 90.000,E1 111.589} C_DIS
LIN {X 0.097,Y -292.260,Z 1906.619,A 0.000,B 0.000,C 90.000,E1 111.354} C_DIS
LIN {X 0.068,Y -296.053,Z 1906.616,A 0.000,B 0.000,C 90.000,E1 110.865} C_DIS
LIN {X 0.061,Y -309.318,Z 1906.603,A 0.000,B 0.000,C 90.000,E1 108.544} C_DIS
LIN {X 0.161,Y -323.891,Z 1906.590,A 0.000,B 0.000,C 90.000,E1 106.260} C_DIS
LIN {X -0.108,Y -337.562,Z 1906.580,A 0.000,B 0.000,C 90.000,E1 104.411} C_DIS
LIN {X 0.039,Y -352.416,Z 1906.570,A 0.000,B 0.000,C 90.000,E1 102.535} C_DIS
LIN {X 0.066,Y -370.794,Z 1906.558,A 0.000,B 0.000,C 90.000,E1 100.489} C_DIS
LIN {X 0.115,Y -389.652,Z 1906.548,A 0.000,B 0.000,C 90.000,E1 98.624} C_DIS
LIN {X 0.033,Y -408.854,Z 1906.539,A 0.000,B 0.000,C 90.000,E1 96.947} C_DIS
LIN {X -0.160,Y -431.222,Z 1906.529,A 0.000,B 0.000,C 90.000,E1 95.220} C_DIS
LIN {X -0.019,Y -439.676,Z 1906.526,A 0.000,B 0.000,C 90.000,E1 94.588} C_DIS
LIN {X -0.061,Y -443.580,Z 1906.523,A 0.000,B 0.000,C 90.000,E1 94.188} C_DIS
LIN {X 0.175,Y -445.263,Z 1906.522,A 0.000,B 0.000,C 90.000,E1 93.898} C_DIS
LIN {X -0.064,Y -446.541,Z 1906.520,A 0.000,B 0.000,C 90.000,E1 93.669} C_DIS
LIN {X -0.113,Y -448.184,Z 1906.517,A 0.000,B 0.000,C 90.000,E1 93.151} C_DIS
LIN {X -0.180,Y -448.797,Z 1906.515,A 0.000,B 0.000,C 90.000,E1 92.636} C_DIS
LIN {X 0.216,Y -448.481,Z 1906.512,A 0.000,B 0.000,C 90.000,E1 92.064} C_DIS
LIN {X 0.181,Y -447.194,Z 1906.509,A 0.000,B 0.000,C 90.000,E1 91.547} C_DIS
LIN {X -0.068,Y -446.125,Z 1906.507,A 0.000,B 0.000,C 90.000,E1 91.318} C_DIS
LIN {X -0.123,Y -443.054,Z 1906.504,A 0.000,B 0.000,C 90.000,E1 90.802} C_DIS
LIN {X 0.207,Y -431.554,Z 1906.494,A 0.000,B 0.000,C 90.000,E1 88.912} C_DIS
LIN {X -0.127,Y -419.792,Z 1906.484,A 0.000,B 0.000,C 90.000,E1 87.078} C_DIS
LIN {X 0.192,Y -408.009,Z 1906.473,A 0.000,B 0.000,C 90.000,E1 85.122} C_DIS
LIN {X -0.140,Y -396.092,Z 1906.462,A 0.000,B 0.000,C 90.000,E1 83.223} C_DIS
LIN {X 0.141,Y -382.434,Z 1906.450,A 0.000,B 0.000,C 90.000,E1 80.914} C_DIS
LIN {X -0.097,Y -368.934,Z 1906.437,A 0.000,B 0.000,C 90.000,E1 78.634} C_DIS
LIN {X 0.088,Y -351.295,Z 1906.419,A 0.000,B 0.000,C 90.000,E1 75.338} C_DIS
LIN {X 0.065,Y -337.698,Z 1906.403,A 0.000,B 0.000,C 90.000,E1 72.598} C_DIS
LIN {X 0.020,Y -325.917,Z 1906.390,A 0.000,B 0.000,C 90.000,E1 70.115} C_DIS
LIN {X 0.065,Y -311.702,Z 1906.372,A 0.000,B 0.000,C 90.000,E1 66.922} C_DIS
LIN {X -0.037,Y -302.195,Z 1906.359,A 0.000,B 0.000,C 90.000,E1 64.665} C_DIS
LIN {X 0.161,Y -290.056,Z 1906.343,A 0.000,B 0.000,C 90.000,E1 61.641} C_DIS
LIN {X -0.091,Y -282.045,Z 1906.331,A 0.000,B 0.000,C 90.000,E1 59.665} C_DIS
LIN {X -0.015,Y -272.555,Z 1906.318,A 0.000,B 0.000,C 90.000,E1 57.248} C_DIS
LIN {X -0.145,Y -264.380,Z 1906.306,A 0.000,B 0.000,C 90.000,E1 55.182} C_DIS
LIN {X -0.081,Y -254.769,Z 1906.293,A 0.000,B 0.000,C 90.000,E1 52.683} C_DIS
LIN {X -0.075,Y -245.175,Z 1906.279,A 0.000,B 0.000,C 90.000,E1 50.150} C_DIS
LIN {X 0.127,Y -234.408,Z 1906.262,A 0.000,B 0.000,C 90.000,E1 47.148} C_DIS
LIN {X -0.114,Y -224.062,Z 1906.245,A 0.000,B 0.000,C 90.000,E1 44.190} C_DIS
LIN {X -0.053,Y -213.022,Z 1906.226,A 0.000,B 0.000,C 90.000,E1 40.701} C_DIS
LIN {X -0.022,Y -205.068,Z 1906.211,A 0.000,B 0.000,C 90.000,E1 37.935} C_DIS
LIN {X -0.044,Y -196.837,Z 1906.193,A 0.000,B 0.000,C 90.000,E1 34.739} C_DIS
LIN {X 0.005,Y -189.336,Z 1906.175,A 0.000,B 0.000,C 90.000,E1 31.465} C_DIS
LIN {X -0.004,Y -182.575,Z 1906.156,A 0.000,B 0.000,C 90.000,E1 28.153} C_DIS
LIN {X 0.049,Y -176.512,Z 1906.138,A 0.000,B 0.000,C 90.000,E1 24.771} C_DIS
LIN {X 0.064,Y -171.278,Z 1906.119,A 0.000,B 0.000,C 90.000,E1 21.354} C_DIS
LIN {X -0.066,Y -166.831,Z 1906.100,A 0.000,B 0.000,C 90.000,E1 17.946} C_DIS
LIN {X 0.025,Y -163.204,Z 1906.080,A 0.000,B 0.000,C 90.000,E1 14.426} C_DIS
LIN {X 0.041,Y -159.519,Z 1906.056,A 0.000,B 0.000,C 90.000,E1 10.018} C_DIS
LIN {X 0.071,Y -157.007,Z 1906.031,A 0.000,B 0.000,C 90.000,E1 5.568} C_DIS
LIN {X -0.028,Y -154.776,Z 1905.997,A 0.000,B 0.000,C 90.000,E1 359.542} C_DIS
LIN {X -0.011,Y -154.134,Z 1905.948,A 0.000,B 0.000,C 90.000,E1 350.557} C_DIS
LIN {X -0.006,Y -156.137,Z 1905.908,A 0.000,B 0.000,C 90.000,E1 343.378} C_DIS
LIN {X 0.028,Y -158.545,Z 1905.883,A 0.000,B 0.000,C 90.000,E1 338.901} C_DIS
LIN {X 0.041,Y -162.153,Z 1905.858,A 0.000,B 0.000,C 90.000,E1 334.460} C_DIS
LIN {X -0.052,Y -166.087,Z 1905.839,A 0.000,B 0.000,C 90.000,E1 330.973} C_DIS
LIN {X 0.045,Y -170.986,Z 1905.819,A 0.000,B 0.000,C 90.000,E1 327.454} C_DIS
LIN {X -0.042,Y -175.304,Z 1905.805,A 0.000,B 0.000,C 90.000,E1 324.895} C_DIS
LIN {X 0.011,Y -180.289,Z 1905.791,A 0.000,B 0.000,C 90.000,E1 322.316} C_DIS
LIN {X 0.011,Y -186.153,Z 1905.777,A 0.000,B 0.000,C 90.000,E1 319.784} C_DIS
LIN {X -0.021,Y -191.755,Z 1905.765,A 0.000,B 0.000,C 90.000,E1 317.715} C_DIS
LIN {X 0.017,Y -199.398,Z 1905.751,A 0.000,B 0.000,C 90.000,E1 315.243} C_DIS
LIN {X -0.080,Y -207.991,Z 1905.738,A 0.000,B 0.000,C 90.000,E1 312.852} C_DIS
LIN {X -0.099,Y -219.072,Z 1905.723,A 0.000,B 0.000,C 90.000,E1 310.092} C_DIS
LIN {X 0.025,Y -231.187,Z 1905.708,A 0.000,B 0.000,C 90.000,E1 307.363} C_DIS
LIN {X -0.156,Y -246.135,Z 1905.691,A 0.000,B 0.000,C 90.000,E1 304.405} C_DIS
LIN {X -0.151,Y -257.985,Z 1905.679,A 0.000,B 0.000,C 90.000,E1 302.212} C_DIS
LIN {X 0.092,Y -272.052,Z 1905.665,A 0.000,B 0.000,C 90.000,E1 299.667} C_DIS
LIN {X -0.132,Y -281.944,Z 1905.655,A 0.000,B 0.000,C 90.000,E1 297.975} C_DIS
LIN {X 0.042,Y -291.547,Z 1905.646,A 0.000,B 0.000,C 90.000,E1 296.232} C_DIS
LIN {X 0.123,Y -296.996,Z 1905.640,A 0.000,B 0.000,C 90.000,E1 295.207} C_DIS
LIN {X 0.126,Y -301.805,Z 1905.635,A 0.000,B 0.000,C 90.000,E1 294.207} C_DIS
LIN {X -0.189,Y -303.935,Z 1905.632,A 0.000,B 0.000,C 90.000,E1 293.770} C_DIS
LIN {X -0.112,Y -314.772,Z 1905.624,A 0.000,B 0.000,C 90.000,E1 292.280} C_DIS
LIN {X 0.066,Y -321.524,Z 1905.618,A 0.000,B 0.000,C 90.000,E1 291.280} C_DIS
LIN {X 0.144,Y -329.745,Z 1905.611,A 0.000,B 0.000,C 90.000,E1 289.993} C_DIS
LIN {X -0.102,Y -337.142,Z 1905.604,A 0.000,B 0.000,C 90.000,E1 288.779} C_DIS
LIN {X 0.060,Y -343.930,Z 1905.597,A 0.000,B 0.000,C 90.000,E1 287.511} C_DIS
LIN {X -0.137,Y -348.440,Z 1905.592,A 0.000,B 0.000,C 90.000,E1 286.622} C_DIS
LIN {X 0.149,Y -352.368,Z 1905.587,A 0.000,B 0.000,C 90.000,E1 285.662} C_DIS
LIN {X 0.034,Y -355.755,Z 1905.582,A 0.000,B 0.000,C 90.000,E1 284.773} C_DIS
LIN {X 0.005,Y -357.725,Z 1905.579,A 0.000,B 0.000,C 90.000,E1 284.175} C_DIS
LIN {X -0.105,Y -359.343,Z 1905.575,A 0.000,B 0.000,C 90.000,E1 283.592} C_DIS
LIN {X -0.202,Y -360.628,Z 1905.572,A 0.000,B 0.000,C 90.000,E1 283.008} C_DIS
LIN {X 0.144,Y -361.493,Z 1905.569,A 0.000,B 0.000,C 90.000,E1 282.355} C_DIS
LIN {X 0.067,Y -361.999,Z 1905.565,A 0.000,B 0.000,C 90.000,E1 281.771} C_DIS
LIN {X -0.004,Y -362.139,Z 1905.562,A 0.000,B 0.000,C 90.000,E1 281.186} C_DIS
LIN {X -0.073,Y -361.839,Z 1905.559,A 0.000,B 0.000,C 90.000,E1 280.602} C_DIS
LIN {X -0.141,Y -361.154,Z 1905.556,A 0.000,B 0.000,C 90.000,E1 280.018} C_DIS
LIN {X 0.143,Y -360.151,Z 1905.552,A 0.000,B 0.000,C 90.000,E1 279.378} C_DIS
LIN {X 0.009,Y -358.813,Z 1905.549,A 0.000,B 0.000,C 90.000,E1 278.803} C_DIS
LIN {X -0.074,Y -357.143,Z 1905.546,A 0.000,B 0.000,C 90.000,E1 278.219} C_DIS
LIN {X 0.084,Y -353.965,Z 1905.541,A 0.000,B 0.000,C 90.000,E1 277.296} C_DIS
LIN {X -0.074,Y -351.401,Z 1905.537,A 0.000,B 0.000,C 90.000,E1 276.720} C_DIS
LIN {X 0.100,Y -348.375,Z 1905.534,A 0.000,B 0.000,C 90.000,E1 276.087} C_DIS
LIN {X -0.087,Y -344.800,Z 1905.531,A 0.000,B 0.000,C 90.000,E1 275.511} C_DIS
LIN {X 0.049,Y -340.568,Z 1905.527,A 0.000,B 0.000,C 90.000,E1 274.878} C_DIS
LIN {X 0.157,Y -335.625,Z 1905.524,A 0.000,B 0.000,C 90.000,E1 274.245} C_DIS
LIN {X -0.026,Y -329.934,Z 1905.520,A 0.000,B 0.000,C 90.000,E1 273.669} C_DIS
LIN {X 0.024,Y -323.730,Z 1905.517,A 0.000,B 0.000,C 90.000,E1 273.094} C_DIS
LIN {X 0.107,Y -317.160,Z 1905.514,A 0.000,B 0.000,C 90.000,E1 272.579} C_DIS
LIN {X -0.068,Y -310.263,Z 1905.512,A 0.000,B 0.000,C 90.000,E1 272.178} C_DIS
LIN {X -0.142,Y -302.782,Z 1905.510,A 0.000,B 0.000,C 90.000,E1 271.833} C_DIS
LIN {X -0.071,Y -294.465,Z 1905.509,A 0.000,B 0.000,C 90.000,E1 271.547} C_DIS
LIN {X 0.105,Y -285.243,Z 1905.508,A 0.000,B 0.000,C 90.000,E1 271.375} C_DIS
LIN {X 0.048,Y -283.049,Z 1905.508,A 0.000,B 0.000,C 90.000,E1 271.375} C_DIS
LIN {X -0.005,Y -181.376,Z 1905.508,A 0.000,B 0.000,C 90.000,E1 271.375} C_DIS
LIN {X -0.023,Y -181.571,Z 1905.503,A 0.000,B 0.000,C 90.000,E1 270.458} C_DIS
LIN {X -0.045,Y -180.906,Z 1905.474,A 0.000,B 0.000,C 90.000,E1 265.412} C_DIS
LIN {X 0.029,Y -180.703,Z 1905.470,A 0.000,B 0.000,C 90.000,E1 264.546} C_DIS
LIN {X -0.069,Y -178.788,Z 1905.442,A 0.000,B 0.000,C 90.000,E1 259.511} C_DIS
LIN {X 0.008,Y -175.835,Z 1905.413,A 0.000,B 0.000,C 90.000,E1 254.393} C_DIS
LIN {X 0.008,Y -172.024,Z 1905.385,A 0.000,B 0.000,C 90.000,E1 249.263} C_DIS
LIN {X -0.016,Y -171.449,Z 1905.380,A 0.000,B 0.000,C 90.000,E1 248.411} C_DIS
LIN {X 0.038,Y -167.684,Z 1905.356,A 0.000,B 0.000,C 90.000,E1 244.076} C_DIS
LIN {X -0.022,Y -166.362,Z 1905.346,A 0.000,B 0.000,C 90.000,E1 242.359} C_DIS
LIN {X -0.029,Y -163.094,Z 1905.327,A 0.000,B 0.000,C 90.000,E1 238.869} C_DIS
LIN {X 0.021,Y -161.038,Z 1905.312,A 0.000,B 0.000,C 90.000,E1 236.215} C_DIS
LIN {X 0.005,Y -157.777,Z 1905.293,A 0.000,B 0.000,C 90.000,E1 232.683} C_DIS
LIN {X 0.068,Y -155.814,Z 1905.278,A 0.000,B 0.000,C 90.000,E1 229.989} C_DIS
LIN {X 0.016,Y -152.066,Z 1905.253,A 0.000,B 0.000,C 90.000,E1 225.526} C_DIS
LIN {X -0.074,Y -150.316,Z 1905.238,A 0.000,B 0.000,C 90.000,E1 222.852} C_DIS
LIN {X -0.052,Y -147.058,Z 1905.213,A 0.000,B 0.000,C 90.000,E1 218.302} C_DIS
LIN {X 0.056,Y -145.636,Z 1905.197,A 0.000,B 0.000,C 90.000,E1 215.518} C_DIS
LIN {X 0.054,Y -143.018,Z 1905.172,A 0.000,B 0.000,C 90.000,E1 210.924} C_DIS
LIN {X -0.015,Y -141.645,Z 1905.151,A 0.000,B 0.000,C 90.000,E1 207.257} C_DIS
LIN {X 0.035,Y -139.441,Z 1905.115,A 0.000,B 0.000,C 90.000,E1 200.737} C_DIS
LIN {X -0.043,Y -139.173,Z 1905.105,A 0.000,B 0.000,C 90.000,E1 198.906} C_DIS
LIN {X -0.015,Y -138.318,Z 1905.053,A 0.000,B 0.000,C 90.000,E1 189.557} C_DIS
LIN {X -0.005,Y -139.471,Z 1905.006,A 0.000,B 0.000,C 90.000,E1 181.146} C_DIS
LIN {X -0.065,Y -141.042,Z 1904.975,A 0.000,B 0.000,C 90.000,E1 175.584} C_DIS
LIN {X 0.030,Y -142.411,Z 1904.960,A 0.000,B 0.000,C 90.000,E1 172.761} C_DIS
LIN {X -0.050,Y -144.646,Z 1904.934,A 0.000,B 0.000,C 90.000,E1 168.173} C_DIS
LIN {X 0.010,Y -147.841,Z 1904.909,A 0.000,B 0.000,C 90.000,E1 163.559} C_DIS
LIN {X -0.047,Y -150.539,Z 1904.888,A 0.000,B 0.000,C 90.000,E1 159.934} C_DIS
LIN {X -0.027,Y -154.005,Z 1904.868,A 0.000,B 0.000,C 90.000,E1 156.305} C_DIS
LIN {X 0.033,Y -157.419,Z 1904.848,A 0.000,B 0.000,C 90.000,E1 152.692} C_DIS
LIN {X 0.055,Y -161.629,Z 1904.829,A 0.000,B 0.000,C 90.000,E1 149.125} C_DIS
LIN {X 0.073,Y -165.825,Z 1904.809,A 0.000,B 0.000,C 90.000,E1 145.595} C_DIS
LIN {X 0.066,Y -170.794,Z 1904.790,A 0.000,B 0.000,C 90.000,E1 142.110} C_DIS
LIN {X -0.017,Y -175.665,Z 1904.771,A 0.000,B 0.000,C 90.000,E1 138.690} C_DIS
LIN {X -0.020,Y -181.279,Z 1904.752,A 0.000,B 0.000,C 90.000,E1 135.283} C_DIS
LIN {X -0.020,Y -186.756,Z 1904.733,A 0.000,B 0.000,C 90.000,E1 131.919} C_DIS
LIN {X 0.052,Y -191.351,Z 1904.719,A 0.000,B 0.000,C 90.000,E1 129.402} C_DIS
LIN {X -0.023,Y -197.188,Z 1904.701,A 0.000,B 0.000,C 90.000,E1 126.137} C_DIS
LIN {X 0.060,Y -200.466,Z 1904.692,A 0.000,B 0.000,C 90.000,E1 124.485} C_DIS
LIN {X 0.077,Y -206.349,Z 1904.674,A 0.000,B 0.000,C 90.000,E1 121.258} C_DIS
LIN {X 0.065,Y -209.625,Z 1904.665,A 0.000,B 0.000,C 90.000,E1 119.667} C_DIS
LIN {X 0.087,Y -216.996,Z 1904.643,A 0.000,B 0.000,C 90.000,E1 115.720} C_DIS
LIN {X 0.040,Y -218.618,Z 1904.639,A 0.000,B 0.000,C 90.000,E1 114.951} C_DIS
LIN {X -0.066,Y -224.142,Z 1904.621,A 0.000,B 0.000,C 90.000,E1 111.844} C_DIS
LIN {X -0.118,Y -283.399,Z 1904.621,A 0.000,B 0.000,C 90.000,E1 111.844} C_DIS
LIN {X 0.041,Y -285.902,Z 1904.621,A 0.000,B 0.000,C 90.000,E1 111.770} C_DIS
LIN {X 0.142,Y -291.624,Z 1904.619,A 0.000,B 0.000,C 90.000,E1 111.408} C_DIS
LIN {X -0.027,Y -294.623,Z 1904.617,A 0.000,B 0.000,C 90.000,E1 111.099} C_DIS
LIN {X -0.062,Y -296.626,Z 1904.615,A 0.000,B 0.000,C 90.000,E1 110.791} C_DIS
LIN {X -0.055,Y -309.773,Z 1904.603,A 0.000,B 0.000,C 90.000,E1 108.489} C_DIS
LIN {X 0.062,Y -324.387,Z 1904.590,A 0.000,B 0.000,C 90.000,E1 106.205} C_DIS
LIN {X 0.128,Y -338.100,Z 1904.580,A 0.000,B 0.000,C 90.000,E1 104.300} C_DIS
LIN {X -0.042,Y -353.000,Z 1904.569,A 0.000,B 0.000,C 90.000,E1 102.479} C_DIS
LIN {X 0.004,Y -371.424,Z 1904.558,A 0.000,B 0.000,C 90.000,E1 100.433} C_DIS
LIN {X 0.115,Y -390.260,Z 1904.548,A 0.000,B 0.000,C 90.000,E1 98.568} C_DIS
LIN {X 0.048,Y -409.511,Z 1904.538,A 0.000,B 0.000,C 90.000,E1 96.891} C_DIS
LIN {X -0.101,Y -431.889,Z 1904.529,A 0.000,B 0.000,C 90.000,E1 95.163} C_DIS
LIN {X 0.074,Y -440.218,Z 1904.525,A 0.000,B 0.000,C 90.000,E1 94.531} C_DIS
LIN {X -0.145,Y -442.261,Z 1904.524,A 0.000,B 0.000,C 90.000,E1 94.359} C_DIS
LIN {X 0.132,Y -444.204,Z 1904.523,A 0.000,B 0.000,C 90.000,E1 94.073} C_DIS
LIN {X -0.003,Y -445.686,Z 1904.521,A 0.000,B 0.000,C 90.000,E1 93.841} C_DIS
LIN {X 0.179,Y -446.868,Z 1904.520,A 0.000,B 0.000,C 90.000,E1 93.555} C_DIS
LIN {X -0.083,Y -447.737,Z 1904.518,A 0.000,B 0.000,C 90.000,E1 93.326} C_DIS
LIN {X -0.123,Y -448.681,Z 1904.516,A 0.000,B 0.000,C 90.000,E1 92.808} C_DIS
LIN {X -0.180,Y -448.679,Z 1904.513,A 0.000,B 0.000,C 90.000,E1 92.293} C_DIS
LIN {X -0.214,Y -447.736,Z 1904.510,A 0.000,B 0.000,C 90.000,E1 91.776} C_DIS
LIN {X 0.182,Y -445.701,Z 1904.507,A 0.000,B 0.000,C 90.000,E1 91.203} C_DIS
LIN {X -0.036,Y -435.949,Z 1904.498,A 0.000,B 0.000,C 90.000,E1 89.656} C_DIS
LIN {X 0.021,Y -425.990,Z 1904.489,A 0.000,B 0.000,C 90.000,E1 88.051} C_DIS
LIN {X 0.121,Y -412.524,Z 1904.477,A 0.000,B 0.000,C 90.000,E1 85.869} C_DIS
LIN {X -0.203,Y -402.370,Z 1904.468,A 0.000,B 0.000,C 90.000,E1 84.261} C_DIS
LIN {X 0.181,Y -390.393,Z 1904.457,A 0.000,B 0.000,C 90.000,E1 82.243} C_DIS
LIN {X -0.024,Y -378.490,Z 1904.446,A 0.000,B 0.000,C 90.000,E1 80.274} C_DIS
LIN {X -0.007,Y -363.449,Z 1904.431,A 0.000,B 0.000,C 90.000,E1 77.645} C_DIS
LIN {X 0.068,Y -346.204,Z 1904.413,A 0.000,B 0.000,C 90.000,E1 74.338} C_DIS
LIN {X 0.119,Y -334.237,Z 1904.399,A 0.000,B 0.000,C 90.000,E1 71.873} C_DIS
LIN {X -0.012,Y -322.531,Z 1904.385,A 0.000,B 0.000,C 90.000,E1 69.390} C_DIS
LIN {X 0.125,Y -309.873,Z 1904.370,A 0.000,B 0.000,C 90.000,E1 66.485} C_DIS
LIN {X -0.020,Y -300.375,Z 1904.357,A 0.000,B 0.000,C 90.000,E1 64.229} C_DIS
LIN {X -0.133,Y -288.298,Z 1904.340,A 0.000,B 0.000,C 90.000,E1 61.257} C_DIS
LIN {X -0.063,Y -278.893,Z 1904.327,A 0.000,B 0.000,C 90.000,E1 58.869} C_DIS
LIN {X 0.082,Y -269.385,Z 1904.314,A 0.000,B 0.000,C 90.000,E1 56.421} C_DIS
LIN {X 0.043,Y -261.164,Z 1904.302,A 0.000,B 0.000,C 90.000,E1 54.322} C_DIS
LIN {X 0.036,Y -251.572,Z 1904.288,A 0.000,B 0.000,C 90.000,E1 51.823} C_DIS
LIN {X -0.069,Y -242.001,Z 1904.274,A 0.000,B 0.000,C 90.000,E1 49.299} C_DIS
LIN {X 0.056,Y -231.354,Z 1904.257,A 0.000,B 0.000,C 90.000,E1 46.296} C_DIS
LIN {X 0.061,Y -221.114,Z 1904.240,A 0.000,B 0.000,C 90.000,E1 43.257} C_DIS
LIN {X 0.035,Y -210.292,Z 1904.221,A 0.000,B 0.000,C 90.000,E1 39.769} C_DIS
LIN {X 0.082,Y -201.564,Z 1904.203,A 0.000,B 0.000,C 90.000,E1 36.583} C_DIS
LIN {X 0.028,Y -193.630,Z 1904.185,A 0.000,B 0.000,C 90.000,E1 33.372} C_DIS
LIN {X 0.061,Y -186.437,Z 1904.167,A 0.000,B 0.000,C 90.000,E1 30.079} C_DIS
LIN {X 0.055,Y -179.962,Z 1904.149,A 0.000,B 0.000,C 90.000,E1 26.744} C_DIS
LIN {X 0.064,Y -175.584,Z 1904.135,A 0.000,B 0.000,C 90.000,E1 24.207} C_DIS
LIN {X 0.055,Y -170.481,Z 1904.116,A 0.000,B 0.000,C 90.000,E1 20.791} C_DIS
LIN {X 0.058,Y -166.183,Z 1904.096,A 0.000,B 0.000,C 90.000,E1 17.330} C_DIS
LIN {X 0.081,Y -162.666,Z 1904.077,A 0.000,B 0.000,C 90.000,E1 13.828} C_DIS
LIN {X 0.065,Y -159.727,Z 1904.057,A 0.000,B 0.000,C 90.000,E1 10.310} C_DIS
LIN {X -0.036,Y -157.137,Z 1904.033,A 0.000,B 0.000,C 90.000,E1 5.910} C_DIS
LIN {X 0.000,Y -154.901,Z 1904.000,A 0.000,B 0.000,C 90.000,E1 360.000} C_DIS
LIN {X -0.011,Y -154.128,Z 1903.948,A 0.000,B 0.000,C 90.000,E1 350.557} C_DIS
LIN {X -0.007,Y -156.133,Z 1903.908,A 0.000,B 0.000,C 90.000,E1 343.378} C_DIS
LIN {X 0.026,Y -158.542,Z 1903.883,A 0.000,B 0.000,C 90.000,E1 338.901} C_DIS
LIN {X 0.040,Y -162.151,Z 1903.858,A 0.000,B 0.000,C 90.000,E1 334.460} C_DIS
LIN {X 0.092,Y -166.090,Z 1903.839,A 0.000,B 0.000,C 90.000,E1 330.923} C_DIS
LIN {X 0.024,Y -169.677,Z 1903.824,A 0.000,B 0.000,C 90.000,E1 328.329} C_DIS
LIN {X -0.040,Y -173.805,Z 1903.810,A 0.000,B 0.000,C 90.000,E1 325.754} C_DIS
LIN {X -0.018,Y -178.550,Z 1903.795,A 0.000,B 0.000,C 90.000,E1 323.176} C_DIS
LIN {X -0.046,Y -184.112,Z 1903.781,A 0.000,B 0.000,C 90.000,E1 320.642} C_DIS
LIN {X 0.029,Y -189.431,Z 1903.770,A 0.000,B 0.000,C 90.000,E1 318.528} C_DIS
LIN {X 0.035,Y -196.760,Z 1903.756,A 0.000,B 0.000,C 90.000,E1 316.053} C_DIS
LIN {X 0.030,Y -205.016,Z 1903.742,A 0.000,B 0.000,C 90.000,E1 313.623} C_DIS
LIN {X -0.052,Y -215.817,Z 1903.727,A 0.000,B 0.000,C 90.000,E1 310.862} C_DIS
LIN {X 0.144,Y -227.614,Z 1903.712,A 0.000,B 0.000,C 90.000,E1 308.096} C_DIS
LIN {X 0.024,Y -242.318,Z 1903.695,A 0.000,B 0.000,C 90.000,E1 305.105} C_DIS
LIN {X -0.029,Y -256.015,Z 1903.681,A 0.000,B 0.000,C 90.000,E1 302.546} C_DIS
LIN {X -0.055,Y -270.034,Z 1903.667,A 0.000,B 0.000,C 90.000,E1 300.050} C_DIS
LIN {X 0.054,Y -280.013,Z 1903.657,A 0.000,B 0.000,C 90.000,E1 298.281} C_DIS
LIN {X 0.075,Y -289.667,Z 1903.648,A 0.000,B 0.000,C 90.000,E1 296.565} C_DIS
LIN {X -0.131,Y -295.235,Z 1903.642,A 0.000,B 0.000,C 90.000,E1 295.591} C_DIS
LIN {X -0.143,Y -300.264,Z 1903.636,A 0.000,B 0.000,C 90.000,E1 294.591} C_DIS
LIN {X 0.128,Y -302.102,Z 1903.635,A 0.000,B 0.000,C 90.000,E1 294.207} C_DIS
LIN {X -0.099,Y -310.577,Z 1903.628,A 0.000,B 0.000,C 90.000,E1 293.078} C_DIS
LIN {X -0.047,Y -319.525,Z 1903.621,A 0.000,B 0.000,C 90.000,E1 291.770} C_DIS
LIN {X 0.051,Y -325.717,Z 1903.616,A 0.000,B 0.000,C 90.000,E1 290.791} C_DIS
LIN {X -0.089,Y -331.488,Z 1903.610,A 0.000,B 0.000,C 90.000,E1 289.866} C_DIS
LIN {X -0.127,Y -340.515,Z 1903.602,A 0.000,B 0.000,C 90.000,E1 288.308} C_DIS
LIN {X 0.082,Y -345.447,Z 1903.596,A 0.000,B 0.000,C 90.000,E1 287.347} C_DIS
LIN {X 0.094,Y -348.451,Z 1903.593,A 0.000,B 0.000,C 90.000,E1 286.732} C_DIS
LIN {X -0.060,Y -352.409,Z 1903.588,A 0.000,B 0.000,C 90.000,E1 285.843} C_DIS
LIN {X -0.172,Y -355.871,Z 1903.583,A 0.000,B 0.000,C 90.000,E1 284.954} C_DIS
LIN {X 0.092,Y -358.746,Z 1903.578,A 0.000,B 0.000,C 90.000,E1 284.008} C_DIS
LIN {X 0.075,Y -360.263,Z 1903.575,A 0.000,B 0.000,C 90.000,E1 283.411} C_DIS
LIN {X -0.016,Y -361.440,Z 1903.571,A 0.000,B 0.000,C 90.000,E1 282.827} C_DIS
LIN {X -0.095,Y -362.215,Z 1903.568,A 0.000,B 0.000,C 90.000,E1 282.243} C_DIS
LIN {X -0.166,Y -362.565,Z 1903.565,A 0.000,B 0.000,C 90.000,E1 281.658} C_DIS
LIN {X 0.193,Y -362.560,Z 1903.561,A 0.000,B 0.000,C 90.000,E1 281.007} C_DIS
LIN {X 0.061,Y -362.160,Z 1903.558,A 0.000,B 0.000,C 90.000,E1 280.433} C_DIS
LIN {X -0.003,Y -361.396,Z 1903.555,A 0.000,B 0.000,C 90.000,E1 279.849} C_DIS
LIN {X -0.072,Y -360.270,Z 1903.551,A 0.000,B 0.000,C 90.000,E1 279.265} C_DIS
LIN {X -0.147,Y -358.787,Z 1903.548,A 0.000,B 0.000,C 90.000,E1 278.681} C_DIS
LIN {X 0.072,Y -357.026,Z 1903.545,A 0.000,B 0.000,C 90.000,E1 278.049} C_DIS
LIN {X -0.120,Y -353.716,Z 1903.540,A 0.000,B 0.000,C 90.000,E1 277.182} C_DIS
LIN {X 0.008,Y -349.512,Z 1903.535,A 0.000,B 0.000,C 90.000,E1 276.258} C_DIS
LIN {X -0.175,Y -346.038,Z 1903.531,A 0.000,B 0.000,C 90.000,E1 275.682} C_DIS
LIN {X -0.030,Y -342.001,Z 1903.528,A 0.000,B 0.000,C 90.000,E1 275.049} C_DIS
LIN {X 0.088,Y -337.401,Z 1903.525,A 0.000,B 0.000,C 90.000,E1 274.416} C_DIS
LIN {X -0.156,Y -331.990,Z 1903.521,A 0.000,B 0.000,C 90.000,E1 273.841} C_DIS
LIN {X 0.052,Y -326.025,Z 1903.518,A 0.000,B 0.000,C 90.000,E1 273.212} C_DIS
LIN {X -0.083,Y -319.567,Z 1903.515,A 0.000,B 0.000,C 90.000,E1 272.694} C_DIS
LIN {X 0.151,Y -312.824,Z 1903.512,A 0.000,B 0.000,C 90.000,E1 272.178} C_DIS
LIN {X 0.135,Y -305.671,Z 1903.510,A 0.000,B 0.000,C 90.000,E1 271.776} C_DIS
LIN {X -0.093,Y -297.865,Z 1903.508,A 0.000,B 0.000,C 90.000,E1 271.489} C_DIS
LIN {X -0.125,Y -293.950,Z 1903.507,A 0.000,B 0.000,C 90.000,E1 271.375} C_DIS
LIN {X -0.102,Y -284.936,Z 1903.507,A 0.000,B 0.000,C 90.000,E1 271.203} C_DIS
LIN {X -0.040,Y -278.544,Z 1903.506,A 0.000,B 0.000,C 90.000,E1 271.146} C_DIS
LIN {X -0.048,Y -181.427,Z 1903.506,A 0.000,B 0.000,C 90.000,E1 271.146} C_DIS
LIN {X 0.036,Y -181.581,Z 1903.501,A 0.000,B 0.000,C 90.000,E1 270.229} C_DIS
LIN {X 0.025,Y -180.894,Z 1903.473,A 0.000,B 0.000,C 90.000,E1 265.179} C_DIS
LIN {X -0.075,Y -179.520,Z 1903.454,A 0.000,B 0.000,C 90.000,E1 261.837} C_DIS
LIN {X 0.087,Y -179.023,Z 1903.445,A 0.000,B 0.000,C 90.000,E1 260.095} C_DIS
LIN {X -0.027,Y -178.660,Z 1903.440,A 0.000,B 0.000,C 90.000,E1 259.285} C_DIS
LIN {X 0.079,Y -175.710,Z 1903.412,A 0.000,B 0.000,C 90.000,E1 254.157} C_DIS
LIN {X 0.088,Y -172.426,Z 1903.388,A 0.000,B 0.000,C 90.000,E1 249.880} C_DIS
LIN {X 0.105,Y -171.251,Z 1903.379,A 0.000,B 0.000,C 90.000,E1 248.156} C_DIS
LIN {X -0.070,Y -167.525,Z 1903.355,A 0.000,B 0.000,C 90.000,E1 243.896} C_DIS
LIN {X 0.012,Y -166.920,Z 1903.350,A 0.000,B 0.000,C 90.000,E1 242.999} C_DIS
LIN {X -0.066,Y -162.915,Z 1903.326,A 0.000,B 0.000,C 90.000,E1 238.663} C_DIS
LIN {X -0.088,Y -161.589,Z 1903.316,A 0.000,B 0.000,C 90.000,E1 236.914} C_DIS
LIN {X 0.038,Y -158.330,Z 1903.296,A 0.000,B 0.000,C 90.000,E1 233.336} C_DIS
LIN {X 0.019,Y -155.632,Z 1903.277,A 0.000,B 0.000,C 90.000,E1 229.784} C_DIS
LIN {X -0.046,Y -151.906,Z 1903.252,A 0.000,B 0.000,C 90.000,E1 225.324} C_DIS
LIN {X -0.030,Y -150.138,Z 1903.237,A 0.000,B 0.000,C 90.000,E1 222.609} C_DIS
LIN {X 0.006,Y -146.925,Z 1903.211,A 0.000,B 0.000,C 90.000,E1 218.051} C_DIS
LIN {X -0.002,Y -145.512,Z 1903.196,A 0.000,B 0.000,C 90.000,E1 215.311} C_DIS
LIN {X -0.007,Y -142.915,Z 1903.171,A 0.000,B 0.000,C 90.000,E1 210.718} C_DIS
LIN {X 0.046,Y -141.536,Z 1903.150,A 0.000,B 0.000,C 90.000,E1 207.001} C_DIS
LIN {X -0.043,Y -139.401,Z 1903.114,A 0.000,B 0.000,C 90.000,E1 200.536} C_DIS
LIN {X -0.038,Y -139.116,Z 1903.104,A 0.000,B 0.000,C 90.000,E1 198.671} C_DIS
LIN {X -0.006,Y -138.353,Z 1903.057,A 0.000,B 0.000,C 90.000,E1 190.254} C_DIS
LIN {X -0.016,Y -139.506,Z 1903.005,A 0.000,B 0.000,C 90.000,E1 180.917} C_DIS
LIN {X 0.066,Y -141.142,Z 1902.974,A 0.000,B 0.000,C 90.000,E1 175.298} C_DIS
LIN {X 0.019,Y -142.522,Z 1902.959,A 0.000,B 0.000,C 90.000,E1 172.534} C_DIS
LIN {X -0.035,Y -144.785,Z 1902.933,A 0.000,B 0.000,C 90.000,E1 167.937} C_DIS
LIN {X -0.048,Y -147.401,Z 1902.912,A 0.000,B 0.000,C 90.000,E1 164.267} C_DIS
LIN {X -0.017,Y -149.976,Z 1902.892,A 0.000,B 0.000,C 90.000,E1 160.604} C_DIS
LIN {X -0.008,Y -153.299,Z 1902.872,A 0.000,B 0.000,C 90.000,E1 156.975} C_DIS
LIN {X -0.020,Y -155.002,Z 1902.862,A 0.000,B 0.000,C 90.000,E1 155.177} C_DIS
LIN {X -0.007,Y -158.644,Z 1902.842,A 0.000,B 0.000,C 90.000,E1 151.591} C_DIS
LIN {X 0.012,Y -161.919,Z 1902.827,A 0.000,B 0.000,C 90.000,E1 148.918} C_DIS
LIN {X 0.037,Y -166.109,Z 1902.808,A 0.000,B 0.000,C 90.000,E1 145.388} C_DIS
LIN {X 0.034,Y -171.119,Z 1902.788,A 0.000,B 0.000,C 90.000,E1 141.904} C_DIS
LIN {X -0.047,Y -175.996,Z 1902.769,A 0.000,B 0.000,C 90.000,E1 138.485} C_DIS
LIN {X 0.066,Y -180.244,Z 1902.755,A 0.000,B 0.000,C 90.000,E1 135.891} C_DIS
LIN {X 0.040,Y -185.658,Z 1902.736,A 0.000,B 0.000,C 90.000,E1 132.528} C_DIS
LIN {X 0.093,Y -190.257,Z 1902.722,A 0.000,B 0.000,C 90.000,E1 130.011} C_DIS
LIN {X -0.017,Y -197.585,Z 1902.700,A 0.000,B 0.000,C 90.000,E1 125.931} C_DIS
LIN {X -0.093,Y -200.847,Z 1902.691,A 0.000,B 0.000,C 90.000,E1 124.326} C_DIS
LIN {X -0.007,Y -206.744,Z 1902.673,A 0.000,B 0.000,C 90.000,E1 121.082} C_DIS
LIN {X -0.012,Y -210.042,Z 1902.664,A 0.000,B 0.000,C 90.000,E1 119.489} C_DIS
LIN {X -0.113,Y -215.818,Z 1902.646,A 0.000,B 0.000,C 90.000,E1 116.360} C_DIS
LIN {X -0.017,Y -219.015,Z 1902.638,A 0.000,B 0.000,C 90.000,E1 114.771} C_DIS
LIN {X -0.078,Y -224.148,Z 1902.621,A 0.000,B 0.000,C 90.000,E1 111.844} C_DIS
LIN {X -0.151,Y -284.296,Z 1902.621,A 0.000,B 0.000,C 90.000,E1 111.844} C_DIS
LIN {X 0.037,Y -288.456,Z 1902.620,A 0.000,B 0.000,C 90.000,E1 111.663} C_DIS
LIN {X 0.058,Y -291.809,Z 1902.619,A 0.000,B 0.000,C 90.000,E1 111.408} C_DIS
LIN {X -0.005,Y -295.470,Z 1902.616,A 0.000,B 0.000,C 90.000,E1 110.972} C_DIS
LIN {X 0.000,Y -312.720,Z 1902.600,A 0.000,B 0.000,C 90.000,E1 108.000} C_DIS
LIN {X 0.085,Y -327.643,Z 1902.588,A 0.000,B 0.000,C 90.000,E1 105.733} C_DIS
LIN {X -0.115,Y -341.639,Z 1902.577,A 0.000,B 0.000,C 90.000,E1 103.883} C_DIS
LIN {X 0.123,Y -356.837,Z 1902.567,A 0.000,B 0.000,C 90.000,E1 102.007} C_DIS
LIN {X 0.092,Y -375.331,Z 1902.556,A 0.000,B 0.000,C 90.000,E1 100.018} C_DIS
LIN {X -0.024,Y -394.286,Z 1902.546,A 0.000,B 0.000,C 90.000,E1 98.219} C_DIS
LIN {X 0.172,Y -416.374,Z 1902.535,A 0.000,B 0.000,C 90.000,E1 96.315} C_DIS
LIN {X 0.003,Y -438.874,Z 1902.526,A 0.000,B 0.000,C 90.000,E1 94.645} C_DIS
LIN {X -0.009,Y -443.072,Z 1902.524,A 0.000,B 0.000,C 90.000,E1 94.245} C_DIS
LIN {X -0.115,Y -444.793,Z 1902.522,A 0.000,B 0.000,C 90.000,E1 94.012} C_DIS
LIN {X 0.191,Y -446.118,Z 1902.521,A 0.000,B 0.000,C 90.000,E1 93.726} C_DIS
LIN {X 0.116,Y -447.957,Z 1902.518,A 0.000,B 0.000,C 90.000,E1 93.212} C_DIS
LIN {X 0.072,Y -448.732,Z 1902.515,A 0.000,B 0.000,C 90.000,E1 92.694} C_DIS
LIN {X 0.017,Y -448.571,Z 1902.512,A 0.000,B 0.000,C 90.000,E1 92.178} C_DIS
LIN {X -0.018,Y -447.457,Z 1902.509,A 0.000,B 0.000,C 90.000,E1 91.661} C_DIS
LIN {X 0.180,Y -446.492,Z 1902.508,A 0.000,B 0.000,C 90.000,E1 91.375} C_DIS
LIN {X -0.068,Y -445.199,Z 1902.506,A 0.000,B 0.000,C 90.000,E1 91.146} C_DIS
LIN {X -0.133,Y -433.714,Z 1902.496,A 0.000,B 0.000,C 90.000,E1 89.312} C_DIS
LIN {X -0.113,Y -423.701,Z 1902.487,A 0.000,B 0.000,C 90.000,E1 87.707} C_DIS
LIN {X -0.148,Y -411.924,Z 1902.477,A 0.000,B 0.000,C 90.000,E1 85.812} C_DIS
LIN {X -0.077,Y -401.758,Z 1902.467,A 0.000,B 0.000,C 90.000,E1 84.147} C_DIS
LIN {X -0.099,Y -389.786,Z 1902.457,A 0.000,B 0.000,C 90.000,E1 82.186} C_DIS
LIN {X 0.127,Y -377.892,Z 1902.445,A 0.000,B 0.000,C 90.000,E1 80.151} C_DIS
LIN {X 0.133,Y -362.868,Z 1902.431,A 0.000,B 0.000,C 90.000,E1 77.521} C_DIS
LIN {X 0.192,Y -345.661,Z 1902.412,A 0.000,B 0.000,C 90.000,E1 74.212} C_DIS
LIN {X 0.126,Y -333.704,Z 1902.399,A 0.000,B 0.000,C 90.000,E1 71.764} C_DIS
LIN {X 0.087,Y -322.009,Z 1902.385,A 0.000,B 0.000,C 90.000,E1 69.263} C_DIS
LIN {X -0.075,Y -309.384,Z 1902.369,A 0.000,B 0.000,C 90.000,E1 66.410} C_DIS
LIN {X 0.052,Y -299.877,Z 1902.356,A 0.000,B 0.000,C 90.000,E1 64.101} C_DIS
LIN {X -0.078,Y -287.824,Z 1902.339,A 0.000,B 0.000,C 90.000,E1 61.129} C_DIS
LIN {X -0.023,Y -278.394,Z 1902.326,A 0.000,B 0.000,C 90.000,E1 58.742} C_DIS
LIN {X 0.108,Y -268.895,Z 1902.313,A 0.000,B 0.000,C 90.000,E1 56.294} C_DIS
LIN {X 0.057,Y -260.669,Z 1902.301,A 0.000,B 0.000,C 90.000,E1 54.196} C_DIS
LIN {X 0.034,Y -251.073,Z 1902.287,A 0.000,B 0.000,C 90.000,E1 51.698} C_DIS
LIN {X 0.071,Y -241.510,Z 1902.273,A 0.000,B 0.000,C 90.000,E1 49.138} C_DIS
LIN {X -0.148,Y -230.876,Z 1902.257,A 0.000,B 0.000,C 90.000,E1 46.215} C_DIS
LIN {X 0.007,Y -220.658,Z 1902.240,A 0.000,B 0.000,C 90.000,E1 43.137} C_DIS
LIN {X -0.012,Y -209.875,Z 1902.220,A 0.000,B 0.000,C 90.000,E1 39.644} C_DIS
LIN {X 0.098,Y -203.264,Z 1902.207,A 0.000,B 0.000,C 90.000,E1 37.237} C_DIS
LIN {X 0.036,Y -195.190,Z 1902.189,A 0.000,B 0.000,C 90.000,E1 34.040} C_DIS
LIN {X -0.059,Y -187.847,Z 1902.171,A 0.000,B 0.000,C 90.000,E1 30.797} C_DIS
LIN {X -0.027,Y -181.231,Z 1902.152,A 0.000,B 0.000,C 90.000,E1 27.462} C_DIS
LIN {X -0.002,Y -175.337,Z 1902.134,A 0.000,B 0.000,C 90.000,E1 24.079} C_DIS
LIN {X -0.017,Y -170.269,Z 1902.115,A 0.000,B 0.000,C 90.000,E1 20.663} C_DIS
LIN {X -0.069,Y -166.007,Z 1902.096,A 0.000,B 0.000,C 90.000,E1 17.221} C_DIS
LIN {X -0.003,Y -162.520,Z 1902.076,A 0.000,B 0.000,C 90.000,E1 13.703} C_DIS
LIN {X -0.054,Y -159.607,Z 1902.057,A 0.000,B 0.000,C 90.000,E1 10.197} C_DIS
LIN {X 0.002,Y -157.058,Z 1902.032,A 0.000,B 0.000,C 90.000,E1 5.739} C_DIS
LIN {X 0.000,Y -154.892,Z 1902.000,A 0.000,B 0.000,C 90.000,E1 360.000} C_DIS
LIN {X -0.012,Y -154.122,Z 1901.948,A 0.000,B 0.000,C 90.000,E1 350.557} C_DIS
